// TwinCAT 3 PLC project JobManagement
// Title: JobManagementFramework
// Company: Bekchoff Automation K.K.
// Author: Takashi Ichihashi
// ProjectVersion: 2.0.0.0
// ProgramVersion: 3.1.4026.21
// CompilerDefines: VISU_USEWSTRING, VISU_NO_EXCEPTION_HANDLING
// libraries:
//   CmpBitmapPool, * (System)
//   Tc2_MC2, * (Beckhoff Automation GmbH)
//   Tc2_Standard, * (Beckhoff Automation GmbH)
//   Tc2_System, * (Beckhoff Automation GmbH)
//   Tc2_Utilities, * (Beckhoff Automation GmbH)
//   Tc3_Module, * (Beckhoff Automation GmbH)
// project tree:
//   DUTs/ ContainerType.TcDUT, ErrorTracking.TcDUT, E_ErrorId.TcDUT, E_FutureExecutionState.TcDUT, ST_JobEventMessage.TcDUT, ST_ModuleCylinder2POS.TcDUT, ST_MotionData.TcDUT
//   / GlobalTextList.TcGTLO, PlcTask.TcTTO, Visualization Manager.TcVMO (not stored), VISU_TASK.TcTTO
//   GVLs/ GVL.TcGVL, ParamFuturesLib.TcGVL
//   POUs/ Command.TcDUT, demo1.TcPOU, demo2.TcPOU, demo3.TcPOU, MotionCommand.TcDUT
//   POUs/model/activities/ FB_EventMessageQueue.TcPOU, FutureCounterBlinkCreator.TcPOU, FutureMCGearIn.TcPOU, FutureMCGearInCreator.TcPOU, FutureMCGearOut.TcPOU, FutureMCGearOutCreator.TcPOU, FutureMCHalt.TcPOU, FutureMCHaltCreator.TcPOU, FutureMCInching.TcPOU, FutureMCInchingCreator.TcPOU, FutureMCMoveAbsolute.TcPOU, FutureMCMoveAbsoluteCreator.TcPOU, FutureMCMoveRelative.TcPOU, FutureMCMoveRelativeCreator.TcPOU, FutureMCMoveVelocity.TcPOU, FutureMCMoveVelocityCreator.TcPOU, FutureMCPower.TcPOU, FutureMCPowerCreator.TcPOU, FutureMCReset.TcPOU, FutureMCResetCreator.TcPOU, FutureMCSetPosition.TcPOU, FutureMCSetPositionCreator.TcPOU, FutureMCStop.TcPOU, FutureMCStopCreator.TcPOU, FutureSleep.TcPOU, FutureSleepCreator.TcPOU, FutureTimerBlink.TcPOU, FutureCounterBlink.TcPOU, FutureTimerBlinkCreator.TcPOU
//   POUs/model/library/ FB_AbstructFuture.TcPOU, FB_BatchJobContainer.TcPOU, FB_BatchJobContainerCreator.TcPOU, FB_AbstructContainer.TcPOU, FB_ParallelJobContainerCreator.TcPOU, FB_ParallelQueueJobContainerCreator.TcPOU, FB_QueueJobContainer.TcPOU, FB_Executor.TcPOU, FB_ParallelJobContainer.TcPOU, FB_ParallelQueueJobContainer.TcPOU, FB_QueueJobContainerCreator.TcPOU, FB_TaskRunner.TcPOU, I_Container.TcIO, I_Future.TcIO, I_SerialContainer.TcIO, I_TaskCreator.TcIO, I_Job.TcIO
//   POUs/model/library/Observer/ FB_JobInfoPublisher.TcPOU (not stored), FB_JobEventLogStr.TcPOU, FB_JobEventCyclicOutput.TcPOU, I_JobInfo.TcIO, I_Observer.TcIO, I_Observable.TcIO
//   POUs/test/ FB_TaskRunner_Test.TcPOU, UnitTest.TcPOU
//   VISUs/ ImagePool.TcIPO (not stored), Visualization.TcVIS
// real-time tasks:
//   TASK PlcTask: cycle T#10ms, priority 10, ADS port 350
//   TASK VISU_TASK: cycle T#100000us, priority 12, ADS port 351
// motion (NC):
//   TASK NC-Task 1 SAF: cycle T#1ms, priority 4, ADS port 501
//   TASK NC-Task 1 SVB: cycle T#10ms, priority 8, ADS port 511
//   AXIS Axis 1 (id 1)
//     OtherSettings: AllowMotionCmdToSlave=true
//     encoder EncType=19
//       EncPara: MaxCount=#xffffffff
//     drive DrvType=16
//       DrvPara: MaxCount=#xffffffff
//         Analog: TorqueSetpointScale=10, ScaleFactorActTorque=0.1
//         TimeComp: TaskDelayCycles=1
//     controller CtrType=1
//       CtrPara: PriorControlFactor=1
//         Observer: BandWidth=20
// I/O:
//   DEVICE Device 1 (EtherCAT) (disabled), AmsNetId 199.4.42.250.2.1
//     Term 1 (EK1100) [EK1100 EtherCAT Coupler (2A E-Bus)]
//       Term 2 (EL2008-0015) [EL2008-0015 8Ch. Dig. Output 24V DC, 0.35A, not short-circuit proof]
//       Term 6 (EL2502) [EL2502 2Ch. PWM output, 24V]
//       Term 5 (EL2596) [EL2596 1-channel LED strobe control terminal 24V/3A]
//       Drive 3 (EL7201-9015) [EL7201-9015 1Ch. DS402 Servo motor output stage with OCT (50V, 2.8A RMS) and STO input]
//       Term 4 (EL9011) [EL9011 End Terminal]
//     Term 7 (EC1100) [EC1100 | EtherCAT coupler, RJ45, angled, push-in]
// variable links:
//   JobManagement/JobManagement Instance <-> NC-Task 1 SAF/Axes/Axis 1
//     PlcTask Inputs/GVL.axis1.NcToPlc <-> Outputs/ToPlc
//     PlcTask Outputs/GVL.axis1.PlcToNc <-> Inputs/FromPlc

CONFIGURATION JobManagement
    RESOURCE PLC ON TwinCAT3
        TASK PlcTask(INTERVAL := T#10ms, PRIORITY := 10);
        TASK VISU_TASK(INTERVAL := T#100000us, PRIORITY := 12);
        PROGRAM demo3 WITH PlcTask : demo3;
        PROGRAM VisuElems_Visu_Prg WITH VISU_TASK : VisuElems.Visu_Prg;
    END_RESOURCE
END_CONFIGURATION

// ---- DUTs/ContainerType.TcDUT
{attribute 'qualified_only'}
{attribute 'strict'}
TYPE ContainerType :
(
	BATCH := 0,
	PARALLEL,
	QUEUE,
	PARALLEL_QUEUE
);
END_TYPE

// ---- DUTs/ErrorTracking.TcDUT
TYPE ErrorTracking :
STRUCT
	job_id : STRING;
	error_id : UDINT;
END_STRUCT
END_TYPE

// ---- DUTs/E_ErrorId.TcDUT
{attribute 'qualified_only'}
{attribute 'strict'}
TYPE E_ErrorId :
(
	PASSIVE_ABORT := 16#FFFFFFFF,
	NOT_CONTAINER := 16#FFFFFFFE
) UDINT;
END_TYPE

// ---- DUTs/E_FutureExecutionState.TcDUT
{attribute 'qualified_only'}
{attribute 'strict'}
{attribute 'to_string'}
TYPE E_FutureExecutionState :
(
	idle := 0,
	init,
	wait_for_process,
	process,
	abort,
	pause,
	quit,
	finish
);
END_TYPE

// ---- DUTs/ST_JobEventMessage.TcDUT
{attribute 'pack_mode' := '1'}
TYPE ST_JobEventMessage :
STRUCT
	subject : T_MaxString;
	job_namespace : T_MaxString;
	job_id : T_MaxString;
	old_state : STRING(16);
	new_state : STRING(16);
	num_of_job : UDINT;
	record_time : ULINT; 
END_STRUCT
END_TYPE

// ---- DUTs/ST_ModuleCylinder2POS.TcDUT
TYPE ST_ModuleCylinder2POS :
STRUCT
	in_pos1	AT%I* : BOOL;
	in_pos2	AT%I* : BOOL;
	out_push AT%Q*	: BOOL;
	out_pull AT%Q*	: BOOL;
	timeout_push	: TIME;	
	timeout_pull	: TIME;	
	current_position : E_2Position := E_2Position.pos1; // pos1 : pull side, pos2: push side
END_STRUCT
END_TYPE

// ---- DUTs/ST_MotionData.TcDUT
TYPE ST_MotionData EXTENDS Tc2_MC2.NCTOPLC_AXIS_REF : 
STRUCT
	record_time : ULINT; 
END_STRUCT
END_TYPE

// ---- POUs/Command.TcDUT
{attribute 'qualified_only'}
{attribute 'strict'}
{attribute 'to_string'}
TYPE Command :
(
	spleep := 0,
	power,
	move_absolute,
	move_relative,
	move_velocity
)UDINT;
END_TYPE

// ---- POUs/MotionCommand.TcDUT
TYPE MotionCommand :
STRUCT
	activate	: BOOL;
	command_id	: Command;
	target		: LREAL;
	velocity	: LREAL;
END_STRUCT
END_TYPE

// ---- GVLs/GVL.TcGVL
{attribute 'qualified_only'}
VAR_GLOBAL
	batch_job_container_creator : FB_BatchJobContainerCreator;
	parallel_job_container_creator : FB_ParallelJobContainerCreator;
	queue_job_container_creator : FB_QueueJobContainerCreator;
	parallel_queue_job_container_creator : FB_ParallelQueueJobContainerCreator;
	axis1	: AXIS_REF;
	axis2	: AXIS_REF;
	motion_command : MotionCommand;
END_VAR

// ---- GVLs/ParamFuturesLib.TcGVL
{attribute 'qualified_only'}
VAR_GLOBAL CONSTANT
	MAX_TASK_NUM : UINT := 40; // Number of max jobs in job container object.
	MAX_STRING_LENGTH : UDINT := 255; // Max string length of task name.
END_VAR

// ---- POUs/model/library/I_Container.TcIO
INTERFACE I_Container EXTENDS __SYSTEM.IQueryInterface

(* This is the generator that iteratively generates references to FB_executor instances*)
METHOD _index_generator_ : UINT;
VAR_INPUT
END_VAR
END_METHOD

METHOD append_job : I_Job
VAR_INPUT
	executor	: I_Job;
END_VAR
END_METHOD

PROPERTY auto_start : BOOL
GET
END_GET
SET
END_SET
END_PROPERTY

PROPERTY continuous_mode : bool
SET
END_SET
END_PROPERTY

METHOD create_container : I_Job
VAR_INPUT
	container_type : ContainerType;
	name: STRING;
END_VAR
END_METHOD

METHOD create_job : I_Job
VAR_INPUT
	creator : I_TaskCreator;
	future_name: STRING;
END_VAR
END_METHOD

PROPERTY each_executor : I_Job
GET
END_GET
END_PROPERTY

PROPERTY num_of_jobs : UDINT
GET
END_GET
END_PROPERTY

METHOD reset : BOOL // Return TRUE if finish.
VAR_INPUT
	deep : BOOL := FALSE;
END_VAR
END_METHOD

METHOD resume : BOOL
VAR_INPUT
END_VAR
END_METHOD

METHOD spawn_job : I_Job
VAR_INPUT
	future : I_Future;
	job_persistence : BOOL := FALSE;
END_VAR
END_METHOD

END_INTERFACE

// ---- POUs/model/library/I_Future.TcIO
{attribute 'enable_dynamic_creation'}
INTERFACE I_Future EXTENDS __System.IQueryInterface

METHOD abort : BOOL // Return TRUE if finish.
VAR_INPUT
END_VAR
END_METHOD

METHOD error_reset : BOOL
VAR_INPUT
END_VAR
END_METHOD

METHOD execute : BOOL // Return TRUE if finish.
VAR_INPUT
END_VAR
END_METHOD

PROPERTY executor : I_Job
GET
END_GET
SET
END_SET
END_PROPERTY

PROPERTY future_name : STRING // Name of future.
GET
END_GET
SET
END_SET
END_PROPERTY

METHOD init : BOOL // Return TRUE if finish.
VAR_INPUT
END_VAR
END_METHOD

PROPERTY nErrorID : HRESULT // Set result code when finished any method. 0 should be set when normal case.
GET
END_GET
END_PROPERTY

PROPERTY persistent_future : BOOL
GET
END_GET
SET
END_SET
END_PROPERTY

METHOD quit : BOOL // Return TRUE if finish.
VAR_INPUT
END_VAR
END_METHOD

PROPERTY state : E_FutureExecutionState // Execution state of this future.
GET
END_GET
SET
END_SET
END_PROPERTY

END_INTERFACE

// ---- POUs/model/library/I_SerialContainer.TcIO
INTERFACE I_SerialContainer EXTENDS __SYSTEM.IQueryInterface

PROPERTY current_job : I_Job
GET
END_GET
END_PROPERTY

END_INTERFACE

// ---- POUs/model/library/I_TaskCreator.TcIO
INTERFACE I_TaskCreator

METHOD create_future : I_Future
VAR_INPUT
	future_name :STRING; // Specify future name
END_VAR
END_METHOD

METHOD destroy_future : I_Future
VAR_INPUT
	future : I_Future; // Specify future instance whtat you want to delete.
END_VAR
END_METHOD

END_INTERFACE

// ---- POUs/model/library/I_Job.TcIO
INTERFACE I_Job EXTENDS __SYSTEM.IQueryInterface

(*abort method

*)
METHOD abort : BOOL // Return TRUE if finish.
VAR_INPUT
END_VAR
END_METHOD

PROPERTY busy : BOOL
GET
END_GET
END_PROPERTY

PROPERTY children : I_Container // Accesser for interface pointer to child container instance.
GET
END_GET
END_PROPERTY

PROPERTY continuous_mode : bool // Make true if keep executing state after all jobs be finished.
SET
END_SET
END_PROPERTY

METHOD create_container : I_Container // Make container object onto child.
VAR_INPUT
	container_type : ContainerType; // specify container type
	name: STRING;	// specify future name
END_VAR
END_METHOD

METHOD create_future : I_Future // Create future dynamically.
VAR_INPUT
	creator : I_TaskCreator; // Specify creator object by which Interface Task Creator implemented.
	future_name: STRING; // Spcfigy future name.
END_VAR
END_METHOD

{attribute 'OPC.UA.DA.Property' := '1'}
{attribute 'monitoring' := 'call'}
{attribute 'OPC.UA.DA.Description' := 'Current state of this executor object.'}
PROPERTY current_state : E_FutureExecutionState // Get current job state
GET
END_GET
END_PROPERTY

PROPERTY current_timestamp : POINTER TO T_FILETIME64
GET
END_GET
SET
END_SET
END_PROPERTY

PROPERTY done : BOOL // Present true if process be finished.
GET
END_GET
END_PROPERTY

METHOD error_reset : BOOL
VAR_INPUT
END_VAR
END_METHOD

METHOD execute : BOOL // Execute future process and return TRUE if all task are finished.
END_METHOD

PROPERTY future : I_Future // Set future instance direct.
GET
END_GET
SET
END_SET
END_PROPERTY

PROPERTY future_creator : I_TaskCreator // Set creator instance.
SET
END_SET
END_PROPERTY

METHOD get_job_info : BOOL
VAR_INPUT
	title		: T_MaxString;
	observable 	: I_Observable;
	recursive	: BOOL := FALSE;
END_VAR
END_METHOD

PROPERTY id : T_MaxString // Get job id.
GET
END_GET
END_PROPERTY

METHOD init : BOOL // Return TRUE if finish.
VAR_INPUT
END_VAR
END_METHOD

PROPERTY job_event_observable : I_Observable
GET
END_GET
SET
END_SET
END_PROPERTY

PROPERTY last_state : E_FutureExecutionState
GET
END_GET
END_PROPERTY

PROPERTY namespace : T_MaxString
GET
END_GET
END_PROPERTY

PROPERTY nErrorID : HRESULT // Present error code when each process,init(), execute(), quit() are finished. '0' represent normal condition without any errors.
GET
END_GET
END_PROPERTY

PROPERTY next_job : I_Job
GET
END_GET
SET
END_SET
END_PROPERTY

PROPERTY parent_executor : I_Job
GET
END_GET
SET
END_SET
END_PROPERTY

PROPERTY persistent_job : BOOL
GET
END_GET
SET
END_SET
END_PROPERTY

PROPERTY previous_job : I_Job
GET
END_GET
SET
END_SET
END_PROPERTY

METHOD quit : BOOL // Return TRUE if finish.
VAR_INPUT
END_VAR
END_METHOD

PROPERTY ready : BOOL
GET
END_GET
END_PROPERTY

METHOD reset : BOOL // Return TRUE if finish.
VAR_INPUT
	deep : BOOL := FALSE;
END_VAR
END_METHOD

METHOD resume : BOOL
END_METHOD

PROPERTY serial : ULINT
GET
END_GET
SET
END_SET
END_PROPERTY

METHOD start : BOOL
END_METHOD

PROPERTY transition : BOOL
GET
END_GET
END_PROPERTY

PROPERTY upstream_aborting : BOOL
GET
END_GET
SET
END_SET
END_PROPERTY

END_INTERFACE

// ---- POUs/model/library/Observer/I_JobInfo.TcIO
INTERFACE I_JobInfo EXTENDS __SYSTEM.IQueryInterface

PROPERTY job : I_Job
GET
END_GET
SET
END_SET
END_PROPERTY

PROPERTY last_state : E_FutureExecutionState
GET
END_GET
SET
END_SET
END_PROPERTY

PROPERTY new_state : E_FutureExecutionState
GET
END_GET
SET
END_SET
END_PROPERTY

PROPERTY record_time : T_FILETIME64
GET
END_GET
SET
END_SET
END_PROPERTY

PROPERTY title : T_MaxString
GET
END_GET
SET
END_SET
END_PROPERTY

END_INTERFACE

// ---- POUs/model/library/Observer/I_Observer.TcIO
INTERFACE I_Observer

METHOD notify : BOOL
VAR_INPUT
	publisher : I_Observable;
END_VAR
END_METHOD

END_INTERFACE

// ---- POUs/model/library/Observer/I_Observable.TcIO
INTERFACE I_Observable  EXTENDS __SYSTEM.IQueryInterface

METHOD add_observer : BOOL
VAR_INPUT
	observer : I_Observer;
END_VAR
END_METHOD

PROPERTY error_id : HRESULT
GET
END_GET
SET
END_SET
END_PROPERTY

METHOD notify_observers : BOOL
END_METHOD

METHOD remove_observer : BOOL
VAR_INPUT
	observer : I_Observer;
END_VAR
END_METHOD

END_INTERFACE

// ---- POUs/demo3.TcPOU
PROGRAM demo3
VAR
	runner : FB_TaskRunner(ContainerType.PARALLEL_QUEUE);

	init: BOOL;
	_state :UINT;
	mc_power : FutureMCPower;
	_handl_power_on	: I_Job;
	_handl_demo_job : I_Job;
	
	_today : TIMESTRUCT;

	bPower : BOOL;
	bStart : BOOL;

	motion_data : ST_MotionData;	
	demo_job_container : FB_BatchJobContainer;
	i : UDINT;
END_VAR

IF NOT init THEN
	JobCreateDemo(demo_job_container, GVL.axis1); // demo_job にメソッドを通してシーケンスジョブを組み立てる
	mc_power.future_name := 'POWER_CTRL';
	init := TRUE;	// RUN 後 1 サイクルだけ実行
END_IF

_today := FILETIME64_TO_SYSTEMTIME(runner.current_time);
runner(root_job_name := 'ROOT',root_job_serial := (_today.wYear MOD 100) * 10000 + _today.wMonth * 100 + _today.wDay);

// Axis
GVL.axis1.ReadStatus();
MEMCPY(ADR(motion_data), ADR(GVL.axis1.NcToPlc), SIZEOF(GVL.axis1.NcToPlc));
motion_data.record_time := runner.current_time;

CASE _state OF
	0:
		IF bPower THEN
			mc_power.set_parameters(axis := GVL.axis1, status := TRUE); // Servo on
			_handl_power_on := runner.append_future(mc_power);
			_state := 1;
		END_IF
	1:
		IF _handl_power_on.ready THEN
			_handl_power_on.start();
		END_IF
		IF _handl_power_on.done THEN
			_state := 2;
		END_IF
	2:
		IF bStart THEN
			_handl_demo_job := runner.append_future(demo_job_container);
			_state := 3;
		END_IF
	3:
		IF _handl_demo_job.ready THEN
			_handl_demo_job.start();
		END_IF
		IF _handl_demo_job.current_state = E_FutureExecutionState.finish THEN
			_state := 2;
			//bStart := FALSE;
		END_IF
		IF NOT bPower THEN
			_state := 4;
		END_IF
	4:
		IF runner.halt(_handl_demo_job) THEN
			_state := 5;
		END_IF
	5:
		mc_power.set_parameters(axis := GVL.axis1, status := FALSE); // Servo off
		_handl_power_on := runner.append_future(mc_power);
		_state := 6;
	6:
		IF _handl_power_on.ready THEN
			_handl_power_on.start();
		END_IF
		IF _handl_power_on.done THEN
			_state := 0;
		END_IF
END_CASE

//IF _state > 0 AND NOT bPower THEN
//END_IF

METHOD JobCreateDemo : BOOL
VAR_INPUT
	job_container : I_Container;
	stAxis1	: REFERENCE TO AXIS_REF;
END_VAR
VAR
	_base_future : I_Future;
	_job_temp : I_Job;
	_job_temp_parent : I_Job;
	sleep : POINTER TO FutureSleep;
	sleep_creator : FutureSleepCreator;

	//mc_move_rel_future : POINTER TO FutureMCMoveRelative;
	mc_move_rel_future_creator : FutureMCMoveRelativeCreator;

	//mc_move_abs_future : POINTER TO FutureMCMoveAbsolute;
	mc_move_abs_future_creator : FutureMCMoveAbsoluteCreator;

	//mc_move_velocity_future: POINTER TO FutureMCMoveVelocity;
	mc_move_velocity_future_creator: FutureMCMoveVelocityCreator;
	
	mc_stop_future_creator : FutureMcStopCreator;
	
	i : UDINT;

END_VAR
//base_job.create_container(ContainerTYpe.BATCH, 'DEMO_JOB');
IF __QUERYINTERFACE(job_container,_base_future) THEN
	_base_future.future_name := 'JOB ROOT';
END_IF

// Sequence
_job_temp_parent := job_container.create_container(ContainerTYpe.BATCH, 'STEP MOVING');
FOR i := 1 TO 4 DO

	mc_move_rel_future_creator.set_parameters(stAxis1,20,200,0,0,0,0);
	_job_temp := _job_temp_parent.children.create_job(mc_move_rel_future_creator,'Move +20 deg, 200 deg/s');

	sleep_creator.sleep_time := T#100MS;
	_job_temp := _job_temp_parent.children.create_job(sleep_creator,'Wait 100ms');
	
END_FOR

// position set to 0

mc_move_abs_future_creator.set_parameters(stAxis1,0,200,0,0,0,0);
_job_temp := job_container.create_job(mc_move_abs_future_creator,'Back to home');

FOR i := 1 TO 10 DO

	mc_move_rel_future_creator.set_parameters(stAxis1,-20,200,0,0,0,0);
	_job_temp := job_container.create_job(mc_move_rel_future_creator,'Move -20 deg, 200 deg/s');

	sleep_creator.sleep_time := T#100MS;
	_job_temp := job_container.create_job(sleep_creator,'Wait 100ms');
	
END_FOR

// position to 0

mc_move_abs_future_creator.set_parameters(stAxis1,0,200,0,0,0,0);
_job_temp := job_container.create_job(mc_move_abs_future_creator,'Back to home');

sleep_creator.sleep_time := T#100MS;
_job_temp := job_container.create_job(sleep_creator,'Wait 100ms');

// 1000deg/s -> 500deg/s

mc_move_velocity_future_creator.set_parameters(stAxis1,MC_Direction.MC_Positive_Direction,10,0,0,0,0);
_job_temp := job_container.create_job(mc_move_velocity_future_creator,'Move velocity');

sleep_creator.sleep_time := T#5S;
_job_temp := job_container.create_job(sleep_creator,'10 deg/s 5 seconds');

mc_move_velocity_future_creator.set_parameters(stAxis1,MC_Direction.MC_Positive_Direction,100,0,0,0,0);
_job_temp := job_container.create_job(mc_move_velocity_future_creator,'Move velocity');

sleep_creator.sleep_time := T#5S;
_job_temp := job_container.create_job(sleep_creator,'100 deg/s 5 seconds');

mc_move_velocity_future_creator.set_parameters(stAxis1,MC_Direction.MC_Positive_Direction,250,0,0,0,0);
_job_temp := job_container.create_job(mc_move_velocity_future_creator,'Move velocity');

sleep_creator.sleep_time := T#5S;
_job_temp := job_container.create_job(sleep_creator,'250 deg/s 5 seconds');

mc_stop_future_creator.set_parameters(stAxis1,0,0);
_job_temp := job_container.create_job(mc_stop_future_creator,'STOP');

// position to 0

mc_move_abs_future_creator.set_parameters(stAxis1,0,250,0,0,0,0);
_job_temp := job_container.create_job(mc_move_abs_future_creator,'Back to home');
END_METHOD

END_PROGRAM

// ---- POUs/model/library/FB_TaskRunner.TcPOU
FUNCTION_BLOCK FB_TaskRunner
VAR_INPUT
	error_reset : BOOL; // Error reset
	root_job_serial : ULINT := 1;
	root_job_name : STRING := 'ROOT';
	upstream_aborting : BOOL := FALSE; // 
	continuous_mode : BOOL := TRUE;
END_VAR
VAR_OUTPUT
	job_empty : BOOL;
	job_namespace : T_MaxString;
	num_of_jobs : UDINT;
END_VAR
VAR
	_executor: FB_Executor; // main Executor
	_observable : FB_JobInfoPublisher;
	last_job_number : UDINT;
	job_event_log_str : FB_JobEventLogStr;	// ジョブイベントをメッセージとしてログ出力するサブスクライバ
	job_event_cyclic_output : FB_JobEventCyclicOutput;	// ADS通信向けにジョブイベントをサイクル単位で出力するためのサブスクライバ
	
	
	fbGetTimeZoneInformation	: FB_GetTimeZoneInformation := (bExecute := TRUE);
	localTime : FB_LocalSystemTime := (bEnable := TRUE);
	tzinfo : FB_GetTimeZoneInformation := (bExecute := TRUE);
	getSystemtime : FB_TzSpecificLocalTimeToSystemTime;
	_current_time : T_FILETIME64;
END_VAR

// 現在時刻の取得
localTime();
tzinfo();
getSystemtime(in := localTime.systemTime, tzInfo := tzinfo.tzInfo);
_current_time := SYSTEMTIME_TO_FILETIME64(getSystemtime.out);
_executor.current_timestamp := ADR(_current_time);

// Job event log for ADS output 
job_event_cyclic_output(); 

_executor.serial := root_job_serial;
_executor.execute();
num_of_jobs := _executor.children.num_of_jobs;

job_empty := last_job_number > 0 AND _executor.children.num_of_jobs = 0;
last_job_number := _executor.children.num_of_jobs;


IF _executor.ready THEN
	_executor.start();
END_IF

METHOD abort : BOOL
VAR_INPUT
	job : I_Job := 0;
END_VAR
VAR
	_child_executor : I_Job;
	all_aborted : BOOL;
END_VAR
IF _executor.children = 0 THEN
	abort := TRUE;
	RETURN;
END_IF

//IF job = 0 OR num_of_jobs = 0 THEN
	all_aborted := TRUE;
//END_IF
REPEAT
	_child_executor := _executor.children.each_executor;
	IF _child_executor <> 0 THEN
		IF job <> 0 THEN
			IF job = _child_executor THEN
				all_aborted := _child_executor.abort();
			END_IF
		ELSE
			IF NOT _child_executor.abort() THEN
				all_aborted := FALSE;
			END_IF
		END_IF

	END_IF
UNTIL
	_child_executor = 0
END_REPEAT

abort := all_aborted;
END_METHOD

METHOD append_future : I_Job
VAR_INPUT
	future : I_Future;
END_VAR
IF _executor.children = 0 THEN
	RETURN;
END_IF

append_future := _executor.children.spawn_job(future, TRUE);
job_namespace := append_future.namespace;
END_METHOD

METHOD append_job : I_Job
VAR_INPUT
	job : I_Job;
END_VAR
IF _executor.children = 0 THEN
	append_job := 0;
	RETURN;
END_IF

append_job := _executor.children.append_job(job);
job_namespace := append_job.namespace;
END_METHOD

METHOD create_job : I_Job
VAR_INPUT
	creator : I_TaskCreator;
	name : STRING;
END_VAR
IF _executor.children = 0 THEN
	RETURN;
END_IF

create_job := _executor.children.create_job(creator, name);
job_namespace := create_job.namespace;
END_METHOD

PROPERTY current_time : T_FILETIME64
GET
current_time := _current_time;
END_GET
END_PROPERTY

METHOD error_reset : BOOL
VAR_INPUT
END_VAR
error_reset := _executor.error_reset();
END_METHOD

//FB_Init is always available implicitly and it is used primarily for initialization.
//The return value is not evaluated. For a specific influence, you can also declare the
//methods explicitly and provide additional code there with the standard initialization
//code. You can evaluate the return value.
METHOD FB_Init: BOOL
VAR_INPUT
    bInitRetains: BOOL; // TRUE: the retain variables are initialized (reset warm / reset cold)
    bInCopyCode: BOOL;  // TRUE: the instance will be copied to the copy code afterward (online change)
	container_type : ContainerType := ContainerType.QUEUE;
END_VAR
_executor.job_event_observable := _observable;
_observable.add_observer(job_event_log_str);
_observable.add_observer(job_event_cyclic_output);
_executor.upstream_aborting := upstream_aborting;
_executor.create_container(container_type, root_job_name);
_executor.continuous_mode := TRUE;
END_METHOD

METHOD halt : BOOL
VAR_INPUT
	job : I_Job;
END_VAR
IF job <> 0 AND_THEN NOT job.done THEN
	IF THIS^.abort(job) THEN
		IF THIS^.quit(job) THEN
			IF THIS^.job_clear(job) THEN
				halt := TRUE;
			END_IF
		END_IF
	END_IF
END_IF
END_METHOD

METHOD job_clear : BOOL
VAR_INPUT
	job : I_Job := 0;
END_VAR
VAR
	_child_executor : I_Job;
	all_clear : BOOL;
	
END_VAR
IF _executor.children = 0 THEN
	job_clear := TRUE;
	RETURN;
END_IF

job_clear := _executor.children.reset(FALSE);
END_METHOD

PROPERTY job_event_observable : I_Observable
GET
job_event_observable := _executor.job_event_observable;
END_GET
SET
_executor.job_event_observable := job_event_observable;
END_SET
END_PROPERTY

METHOD quit : BOOL
VAR_INPUT
	job : I_Job := 0;
END_VAR
VAR
	_child_executor : I_Job;
	all_quit: BOOL;
END_VAR
IF _executor.children = 0 THEN
	quit := TRUE;
	RETURN;
END_IF

//IF job = 0 OR _executor.children.num_of_jobs > 0 THEN
	all_quit := TRUE;
//END_IF

REPEAT
	_child_executor := _executor.children.each_executor;
	IF _child_executor <> 0 THEN
		IF job <> 0 THEN
			IF job = _child_executor THEN
				all_quit := _child_executor.quit();
			END_IF
		ELSE
			IF NOT _child_executor.quit() THEN
				all_quit := FALSE;
			END_IF
		END_IF

	END_IF
UNTIL
	_child_executor = 0
END_REPEAT

quit := all_quit;
END_METHOD

METHOD restart : BOOL
VAR_INPUT
END_VAR
IF _executor.error_reset() THEN
	restart := _executor.resume();
END_IF
END_METHOD

PROPERTY root_executor : I_Job
GET
root_executor := _executor;
END_GET
END_PROPERTY

END_FUNCTION_BLOCK

// ---- POUs/model/library/FB_Executor.TcPOU
{attribute 'enable_dynamic_creation'}
FUNCTION_BLOCK FB_Executor IMPLEMENTS I_Job
VAR_INPUT
END_VAR
VAR_OUTPUT
END_VAR
VAR
	{attribute 'TcEncoding':='UTF-8'}
	_namespace : T_MaxString;
	_id : T_MaxString;
	_done : BOOL;
	_start : BOOL;
	_resume : BOOL;
	_passive_abort : BOOL;
	_quit : BOOL;
	_upstream_aborting : BOOL := FALSE;
	 {attribute 'TcAnalytics'}
	 _state :E_FutureExecutionState := E_FutureExecutionState.idle;
	_last_state  :E_FutureExecutionState;
	_error_id : HRESULT;
	_aborting :BOOL;
	_quitting :BOOL;
	_interface_container : I_Container := 0;
	_job_event_observable : I_Observable;
	_future_creator : I_TaskCreator;
	_future : I_Future;
	_parent_job : I_Job := 0;
	_persistent_job : BOOL := TRUE;
	_current_timestamp : POINTER TO T_FILETIME64 := 0;
	_previous_job : I_Job;
	_next_job : I_Job;
	_transition : BOOL;
END_VAR
VAR PERSISTENT
	_serial	: ULINT;
END_VAR

(*abort method

*)
METHOD abort : BOOL // Return TRUE if finish.
VAR_INPUT
END_VAR
IF _state = E_FutureExecutionState.init OR
   _state = E_FutureExecutionState.process OR
   _state = E_FutureExecutionState.quit THEN
   	_start := FALSE;
	_passive_abort := TRUE;
	abort := FALSE;
ELSE
	IF _state = E_FutureExecutionState.abort THEN
		abort := NOT _aborting;
	ELSE
		abort := TRUE;
	END_IF
END_IF
THIS^.execute();
END_METHOD

PROPERTY busy : BOOL
GET
busy := (	_state = E_FutureExecutionState.init OR	
			_state = E_FutureExecutionState.process OR 
			_state = E_FutureExecutionState.quit
		);
END_GET
END_PROPERTY

PROPERTY children : I_Container // Accesser for interface pointer to child container instance.
GET
children := _interface_container;
END_GET
END_PROPERTY

PROPERTY continuous_mode : bool // Make true if keep executing state after all jobs be finished.
SET
IF _interface_container <> 0 THEN
	_interface_container.continuous_mode := continuous_mode;
END_IF
END_SET
END_PROPERTY

METHOD create_container : I_Container // Make container object onto child.
VAR_INPUT
	container_type : ContainerType; // specify container type
	name: STRING;	// specify future name
END_VAR
VAR
	delete_existing_container : BOOL;
	created_future : I_Future;
END_VAR
IF _interface_container <> 0 THEN
 	IF _interface_container.reset(FALSE) THEN
		delete_existing_container := TRUE;
	ELSE
		delete_existing_container := FALSE;
	END_IF
ELSE
	delete_existing_container := TRUE;
END_IF

IF delete_existing_container THEN
	CASE container_type OF
		ContainerType.BATCH:
			created_future := create_future(GVL.batch_job_container_creator, name);
			created_future.executor.persistent_job := FALSE;
		ContainerType.PARALLEL:
			created_future := create_future(GVL.parallel_job_container_creator, name);
			created_future.executor.persistent_job := FALSE;
		ContainerType.QUEUE:
			created_future := create_future(GVL.queue_job_container_creator, name);
			created_future.executor.persistent_job := TRUE;
		ContainerType.PARALLEL_QUEUE:
			created_future := create_future(GVL.parallel_queue_job_container_creator, name);
			created_future.executor.persistent_job := TRUE;
	END_CASE
	THIS^.init();
	create_container := THIS^.children;
END_IF
END_METHOD

METHOD create_future : I_Future // Create future dynamically.
VAR_INPUT
	creator : I_TaskCreator; // Specify creator object by which Interface Task Creator implemented.
	future_name: STRING; // Spcfigy future name.
END_VAR
_future_creator := creator;
IF _future_creator <> 0 THEN
	THIS^.future := creator.create_future(future_name);
	_future.persistent_future := FALSE;
END_IF
create_future := _future;
END_METHOD

{attribute 'OPC.UA.DA.Property' := '1'}
{attribute 'monitoring' := 'call'}
{attribute 'OPC.UA.DA.Description' := 'Current state of this executor object.'}
PROPERTY current_state : E_FutureExecutionState // Get current job state
GET
current_state := _state;
END_GET
END_PROPERTY

PROPERTY current_timestamp : POINTER TO T_FILETIME64
GET
current_timestamp := _current_timestamp;
END_GET
SET
_current_timestamp := current_timestamp;
END_SET
END_PROPERTY

PROPERTY done : BOOL // Present true if process be finished.
GET
done := _done;
END_GET
END_PROPERTY

METHOD error_reset : BOOL
VAR_INPUT
END_VAR
IF _future <> 0 THEN
	IF _future.error_reset() THEN
		error_reset := TRUE;
		get_job_info('ERROR_RESET', _job_event_observable, FALSE);
	ELSE
		error_reset := FALSE;
	END_IF
	_error_id := _future.nErrorID;
ELSE
	_error_id := 0;
	error_reset := TRUE;
END_IF
END_METHOD

METHOD execute : BOOL // Execute future process and return TRUE if all task are finished.
VAR_INST
	_state_mem :E_FutureExecutionState;
	delay : TIME := T#3S;
	sleep : TON;
	await : BOOL;
	_logging : BOOL;
END_VAR
VAR
	_executor : REFERENCE TO FB_Executor;
	start_all_children : BOOL;
	exe: INT;
END_VAR
IF _future = 0 THEN
	execute := TRUE;
	RETURN;
ELSE
	execute := FALSE;
END_IF

IF _passive_abort THEN
	_state := E_FutureExecutionState.abort;
	//IF _error_id = 0 THEN
	//	_error_id := E_ErrorId.PASSIVE_ABORT;
	//END_IF
	_passive_abort := FALSE;
END_IF

IF _quit THEN
	_state := E_FutureExecutionState.quit;
END_IF
_quit := FALSE;

CASE _state OF
	E_FutureExecutionState.idle:
		IF _future.state = E_FutureExecutionState.idle OR 
			_future.state = E_FutureExecutionState.finish THEN
			IF init() THEN
				_state := E_FutureExecutionState.init;
			END_IF
		END_IF
	E_FutureExecutionState.init:
		IF _future.init() THEN
			IF _future.nErrorID = 0 THEN
				_state := E_FutureExecutionState.wait_for_process;
			ELSE
				_last_state := E_FutureExecutionState.init;
				_error_id := _future.nErrorID;
				_state := E_FutureExecutionState.abort;
			END_IF
		END_IF
	E_FutureExecutionState.wait_for_process: 
		IF _start THEN
			IF _previous_job <> 0 AND_THEN _future <> 0 AND_THEN _previous_job.future = _future THEN
				IF _future.init() THEN
					_state := E_FutureExecutionState.process;
					_start := FALSE;					
				END_IF
			ELSE
				_state := E_FutureExecutionState.process;
				_start := FALSE;
			END_IF
		END_IF
	E_FutureExecutionState.process: 
		IF _future.execute() THEN
			IF _future.nErrorID = 0 THEN
				_state := E_FutureExecutionState.quit;
				_done := TRUE;
			ELSE
				_error_id := _future.nErrorID;
				_state := E_FutureExecutionState.abort;
			END_IF
		END_IF
	E_FutureExecutionState.abort:
		IF _aborting THEN
			await := _future.abort();
			_resume := FALSE;
			IF _upstream_aborting AND _parent_job <> 0 THEN
				_parent_job.abort();
			END_IF
			IF await THEN
				_aborting := FALSE;
			END_IF
		ELSIF _resume THEN
			_state := _last_state;
			IF _error_id = E_ErrorId.PASSIVE_ABORT THEN
				_error_id := 0;
			END_IF
			_resume := FALSE;
		END_IF
	E_FutureExecutionState.quit:
		IF _future.quit() THEN
			IF _future.nErrorID = 0 THEN
				_state := E_FutureExecutionState.finish;
			ELSE
				_error_id := _future.nErrorID;
				_state := E_FutureExecutionState.abort;
			END_IF
			_quitting := FALSE;
		END_IF
	E_FutureExecutionState.finish:
		IF NOT _logging THEN
			execute := TRUE;
		END_IF
END_CASE

IF _state <> _state_mem THEN
	_last_state := _state_mem;

	IF _state = E_FutureExecutionState.init OR
		_state = E_FutureExecutionState.process OR
		_state = E_FutureExecutionState.quit THEN
		_error_id := 0;
	END_IF

	IF _state = E_FutureExecutionState.abort THEN
		_aborting := TRUE;
	END_IF
	
	IF _state = E_FutureExecutionState.quit THEN
		sleep(IN := FALSE);
		_quitting := TRUE;
	END_IF

	_logging := TRUE;

END_IF

_transition := _state <> _state_mem;
_state_mem := _state;

// Transition logging
IF _logging THEN
	IF get_job_info('TRANSITION', _job_event_observable,FALSE) THEN
		_logging := FALSE;
	END_IF
END_IF



IF _future <> 0 THEN
	_future.state := _state;
END_IF
END_METHOD

PROPERTY future : I_Future // Set future instance direct.
GET
future := _future;
END_GET
SET
VAR
	_eval_executor : I_Job;
END_VAR
_future := future;
_future.state := _state;
_future.executor := THIS^;
//_future.persistent_future := TRUE;
IF NOT __QUERYINTERFACE(_future, _interface_container) THEN
	_interface_container := 0;
END_IF

_future.persistent_future := TRUE;

// Redefine parent job pointer to the container members which has been set as the new future.
IF _interface_container <> 0 THEN
	REPEAT
		_eval_executor := _interface_container.each_executor;
		IF _eval_executor <> 0 THEN
			// Set persistent future flag when redefine new parent due to make bound of namespace.
			//IF _eval_executor.parent_executor = 0 AND _eval_executor.children <> 0 THEN
			//	_eval_executor.future.persistent_future := TRUE;
			//END_IF
			// Set new parent for each childrens
			_eval_executor.parent_executor := THIS^;
		END_IF
	UNTIL
		_eval_executor = 0
	END_REPEAT
END_IF
END_SET
END_PROPERTY

PROPERTY future_creator : I_TaskCreator // Set creator instance.
SET
_future_creator := future_creator;
END_SET
END_PROPERTY

METHOD get_job_info : BOOL
VAR_INPUT
	title		: T_MaxString; // Observable object title
	observable 	: I_Observable; // Observable object
	recursive	: BOOL := FALSE; // Set observable to child job recursively or not
END_VAR
VAR
	_info : I_JobInfo;
	_child_job : I_Job;
	_cmp : BOOL;
END_VAR
IF observable = 0  OR NOT __QUERYINTERFACE(observable, _info) THEN
	get_job_info := TRUE;
	RETURN;
END_IF

_info.title := title;
_info.job := THIS^;
_info.last_state := _last_state;
_info.new_state := _state;
IF _current_timestamp <> 0 THEN
	_info.record_time := _current_timestamp^;
ELSE
	_info.record_time := F_GetSystemTime();
END_IF

observable.notify_observers();

IF recursive THEN
	_cmp := TRUE;
	IF THIS^.children <> 0 THEN
		REPEAT
			_child_job := THIS^.children.each_executor;
			IF _child_job <> 0 THEN
				IF NOT _child_job.get_job_info(title, observable, recursive) THEN
					_cmp := FALSE;
				END_IF
			END_IF
		UNTIL
			_child_job = 0
		END_REPEAT
	END_IF
	
	get_job_info := _cmp;
ELSE
	get_job_info := TRUE;
END_IF
END_METHOD

PROPERTY id : T_MaxString // Get job id.
GET
id := _id;
END_GET
END_PROPERTY

METHOD init : BOOL // Return TRUE if finish.
VAR_INPUT
END_VAR
VAR
	_eval_executor : I_Job;
END_VAR
_done := FALSE;
_passive_abort := FALSE;
_start := FALSE;
_state := E_FutureExecutionState.idle;
_error_id := 0;

_eval_executor := _parent_job;
_id := CONCAT('/', TO_STRING(_serial));
REPEAT
	IF _eval_executor <> 0 THEN
		_id := CONCAT(TO_STRING(_eval_executor.serial), _id);
		_id := CONCAT('/',_id);
		_eval_executor := _eval_executor.parent_executor;
	END_IF
UNTIL
	_eval_executor = 0
END_REPEAT


IF _parent_job = 0 THEN
	_namespace := _id;
ELSIF _future <> 0 AND_THEN _future.persistent_future AND_THEN NOT _parent_job.future.persistent_future THEN
	_namespace := _id;
ELSE
	_namespace := _parent_job.namespace;
END_IF

INIT := TRUE;
END_METHOD

PROPERTY job_event_observable : I_Observable
GET
job_event_observable := _job_event_observable;
END_GET
SET
VAR
	executor : I_Job;
END_VAR
_job_event_observable := job_event_observable;
IF THIS^.children <> 0 THEN
	REPEAT
		executor := THIS^.children.each_executor;
		IF executor <> 0 THEN
			executor.job_event_observable := job_event_observable;
		END_IF
	UNTIL
		executor = 0
	END_REPEAT
END_IF
END_SET
END_PROPERTY

PROPERTY last_state : E_FutureExecutionState
GET
last_state := _last_state;
END_GET
END_PROPERTY

PROPERTY namespace : T_MaxString
GET
namespace := _namespace;
END_GET
END_PROPERTY

PROPERTY nErrorID : HRESULT // Present error code when each process,init(), execute(), quit() are finished. '0' represent normal condition without any errors.
GET
nErrorID := _error_id;
END_GET
END_PROPERTY

PROPERTY next_job : I_Job
GET
next_job := _next_job;
END_GET
SET
_next_job := next_job;
END_SET
END_PROPERTY

PROPERTY parent_executor : I_Job
GET
parent_executor := _parent_job;
END_GET
SET
VAR
END_VAR
VAR
	_parent_path : T_MaxString;
END_VAR
_parent_job := parent_executor;
THIS^.current_timestamp := _parent_job.current_timestamp;
END_SET
END_PROPERTY

PROPERTY persistent_job : BOOL
GET
persistent_job := _persistent_job;
END_GET
SET
_persistent_job := persistent_job;
END_SET
END_PROPERTY

PROPERTY previous_job : I_Job
GET
previous_job := _previous_job;
END_GET
SET
_previous_job := previous_job;
END_SET
END_PROPERTY

METHOD quit : BOOL // Return TRUE if finish.
VAR_INPUT
END_VAR
IF _state = E_FutureExecutionState.init OR
   _state = E_FutureExecutionState.process OR
   _state = E_FutureExecutionState.quit THEN
	_quit := TRUE;	
END_IF

IF 	_quit AND _state = E_FutureExecutionState.quit THEN
	quit := NOT _quitting;
ELSE
	quit := TRUE;
END_IF
END_METHOD

PROPERTY ready : BOOL
GET
ready := _state = E_FutureExecutionState.wait_for_process;
END_GET
END_PROPERTY

METHOD reset : BOOL // Return TRUE if finish.
VAR_INPUT
	deep : BOOL := FALSE;
END_VAR
VAR
	_reset_children :BOOL := FALSE;
END_VAR
// Waiting finish process and remove jobs from container items.
IF THIS^.busy THEN
	THIS^.abort();
ELSIF _interface_container <> 0 AND _future <> 0 AND_THEN 
	( NOT _future.persistent_future OR deep) THEN
	_reset_children := _interface_container.reset(deep);
ELSE
	_reset_children := TRUE;
END_IF

// Remove my future.
IF _reset_children AND _future <> 0 THEN
	IF  NOT _future.persistent_future OR deep THEN
		IF _future_creator <> 0 THEN
			_future := _future_creator.destroy_future(_future);
		ELSIF _future.init() THEN
			_future.state := E_FutureExecutionState.idle;
			_future := 0;
		END_IF
		IF _future = 0 THEN
			_interface_container := 0;
			reset := TRUE;
		END_IF
	ELSE
		IF _future.init() THEN
			reset := TRUE;
		END_IF
	END_IF
END_IF
END_METHOD

METHOD resume : BOOL
VAR_INST
	_executor : REFERENCE TO FB_Executor;
END_VAR
_resume := TRUE;
IF _interface_container <> 0 THEN
	IF NOT _interface_container.resume() THEN
		_resume := FALSE;
	END_IF
END_IF
IF NOT _resume THEN
	_future.execute();
END_IF
resume := _resume;
END_METHOD

PROPERTY serial : ULINT
GET
serial := _serial;
END_GET
SET
_serial := serial;
END_SET
END_PROPERTY

METHOD start : BOOL
VAR
	_start_children :BOOL := FALSE;
END_VAR
// Start my future.
_start := _state = E_FutureExecutionState.wait_for_process;
start := TRUE;
END_METHOD

PROPERTY transition : BOOL
GET
transition := _transition;
END_GET
END_PROPERTY

PROPERTY upstream_aborting : BOOL
GET
upstream_aborting := _upstream_aborting;
END_GET
SET
_upstream_aborting := upstream_aborting;
END_SET
END_PROPERTY

END_FUNCTION_BLOCK

// ---- POUs/model/library/Observer/FB_JobEventLogStr.TcPOU
FUNCTION_BLOCK FB_JobEventLogStr IMPLEMENTS I_Observer

METHOD notify : BOOL
VAR_INPUT
	publisher	: I_Observable;
END_VAR
VAR_INST
	fb_timezone_info : FB_GetTimeZoneInformation := (bExecute := TRUE);
	text : T_MaxString;
END_VAR
VAR
	job_info : I_JobInfo;
	container : I_Container;
	num_of_jobs : UDINT;
END_VAR

IF NOT __QUERYINTERFACE(publisher, job_info) THEN
	RETURN;
END_IF

IF job_info.job.children <> 0 THEN
	num_of_jobs := job_info.job.children.num_of_jobs;
ELSE
	num_of_jobs := 0;
END_IF

IF job_info.job <> 0 THEN
	text := '';
	//fb_timezone_info();
	//text := FILETIME64_TO_ISO8601(fileTime := job_report.record_time, nBias := DINT_TO_INT(fb_timezone_info.tzInfo.bias), bUTC := TRUE,nPrecision := 6);
	//text := CONCAT(text, ' ');
	//text := CONCAT(text, job_report.title);
	text := CONCAT(text, '		');
	text := CONCAT(text, job_info.job.id);
	text := CONCAT(text, '		');
	text := CONCAT(text, job_info.job.namespace);
	text := CONCAT(text, '		');
	text := CONCAT(text, TO_STRING(num_of_jobs));
	text := CONCAT(text, '		');
	text := CONCAT(text, TO_STRING(job_info.new_state));
	text := CONCAT(text, '		');
	text := CONCAT(text, TO_STRING(job_info.job.nErrorID));
	text := CONCAT(text, '		');
	text := CONCAT(text, job_info.job.future.future_name);
	
	ADSLOGSTR(msgCtrlMask := ADSLOG_MSGTYPE_LOG,
 			 msgFmtStr := text, 
			strArg := '');	
END_IF

notify := TRUE;
END_METHOD

END_FUNCTION_BLOCK

// ---- POUs/model/library/Observer/FB_JobEventCyclicOutput.TcPOU
FUNCTION_BLOCK FB_JobEventCyclicOutput IMPLEMENTS I_Observer
VAR_OUTPUT
	event_message : ST_JobEventMessage;
END_VAR
VAR
	queue : FB_EventMessageQueue;
	cycle_counter : UINT;
END_VAR

IF queue.usage > 0 THEN
	event_message := queue.get();
END_IF

METHOD notify : BOOL
VAR_INPUT
	publisher	: I_Observable;
END_VAR
VAR_INST
	_event_message : ST_JobEventMessage;
END_VAR
VAR
	job_info : I_JobInfo;
	container : I_Container;
	num_of_jobs : UDINT;
END_VAR
IF NOT __QUERYINTERFACE(publisher, job_info) THEN
	RETURN;
END_IF

IF job_info.job.children <> 0 THEN
	num_of_jobs := job_info.job.children.num_of_jobs;
ELSE
	num_of_jobs := 0;
END_IF

_event_message.job_id := job_info.job.id;
_event_message.job_namespace := job_info.job.namespace;
_event_message.num_of_job := num_of_jobs;
_event_message.new_state := TO_STRING(job_info.new_state);
_event_message.old_state := TO_STRING(job_info.last_state);
_event_message.record_time := job_info.record_time;
_event_message.subject := job_info.job.future.future_name;
queue.put(_event_message);
notify := TRUE;
END_METHOD

END_FUNCTION_BLOCK

// ---- POUs/model/activities/FB_EventMessageQueue.TcPOU
FUNCTION_BLOCK FB_EventMessageQueue
VAR CONSTANT
	COMMAND_QUEUE_BUFFER_SIZE :UDINT := 50;
END_VAR
VAR_OUTPUT
END_VAR
VAR
	_usage:	UDINT;
	_write_index : UDINT := 1;
	_read_index : UDINT := 1;
	_queue_size:	UDINT := COMMAND_QUEUE_BUFFER_SIZE;
	queue_buffer:	ARRAY [1..COMMAND_QUEUE_BUFFER_SIZE] OF ST_JobEventMessage;
END_VAR

PROPERTY full : BOOL
GET
full :=  _usage >= COMMAND_QUEUE_BUFFER_SIZE;
END_GET
END_PROPERTY

METHOD get : REFERENCE TO ST_JobEventMessage
VAR_INPUT
END_VAR
IF _usage = 0 THEN
	get REF= 0;
	RETURN;
END_IF

get REF= queue_buffer[_read_index];

_usage := _usage - 1;

IF COMMAND_QUEUE_BUFFER_SIZE > _read_index THEN
	_read_index := _read_index + 1;
ELSE
	_read_index := 1;
END_IF
END_METHOD

METHOD put : BOOL
VAR_INPUT
	fbEvent:	REFERENCE TO ST_JobEventMessage;
END_VAR
IF _usage >= COMMAND_QUEUE_BUFFER_SIZE THEN
	put := FALSE;
ELSE
	queue_buffer[_write_index] := fbEvent;
	_usage := _usage + 1;
	IF COMMAND_QUEUE_BUFFER_SIZE > _write_index THEN
		_write_index := _write_index + 1;
	ELSE
		_write_index := 1;
	END_IF
	put := TRUE;
END_IF
END_METHOD

PROPERTY usage : UDINT
GET
usage := _usage;
END_GET
END_PROPERTY

END_FUNCTION_BLOCK

// ---- POUs/model/activities/FutureMCPower.TcPOU
{attribute 'enable_dynamic_creation'}
FUNCTION_BLOCK FutureMCPower EXTENDS FB_AbstructFuture
VAR_INPUT
END_VAR
VAR_OUTPUT
END_VAR
VAR
	_axis: REFERENCE TO AXIS_REF;
	_override: LREAL := 100.0;
	_enable_positive:	BOOL := TRUE; 
	_enable_negative:	BOOL := TRUE;
	_fb_power	: MC_Power;
	_mc_reset	: MC_Reset;
	_mc_stop	: MC_Stop;
	_option : ST_PowerOptions;
	_buffer_mode : MC_BufferMode;
	_status : BOOL;
END_VAR

METHOD error_reset : BOOL // Must be overrided if future has any errors.
VAR_INST
	_exec_state : UDINT;
END_VAR
IF _error_id <> 0 THEN
	CASE _exec_state OF
		0:
			_mc_reset(Axis := _axis, Execute := FALSE);
			_mc_reset(Axis:= _axis, Execute := TRUE );
			_exec_state := 1;
		1:
			IF _mc_reset.Busy THEN
				_mc_reset(Axis:= _axis,Execute := FALSE);
				error_reset := TRUE;
			END_IF
	END_CASE	
	_error_id := _fb_power.ErrorID;
ELSE
	error_reset := TRUE;
END_IF
END_METHOD

METHOD execute : BOOL // Return TRUE if finish.
VAR_INST
	_exec_state: UINT;
	_stoped : BOOL;
END_VAR
_axis.ReadStatus();
IF _axis.Status.Moving THEN
	_stoped := FALSE;
	_exec_state := 0;
END_IF

IF NOT _stoped THEN
	CASE _exec_state OF
		0:
			_mc_stop(axis := _axis, Execute := FALSE);
			_mc_stop(
				Axis:= _axis,
				Execute := TRUE
			);
			_exec_state := 1;
		1:
			IF _mc_stop.Busy THEN
				_mc_stop(Axis:= _axis,Execute := FALSE);
				_stoped := TRUE;
			END_IF
	END_CASE
END_IF
	
IF _axis.Status.NotMoving AND _stoped THEN
	_fb_power(
		Axis:= _axis, 
		Enable:= _status, 
		Enable_Positive:= _enable_positive, 
		Enable_Negative:= _enable_negative, 
		Override:= _override, 
		BufferMode:= _buffer_mode, 
		Options:= _option, 
	);
	_error_id := _fb_power.ErrorID;
	execute := _status = _fb_Power.Status;
END_IF
END_METHOD

METHOD set_options : BOOL
VAR_INPUT
	Enable_Positive:	BOOL; 
	Enable_Negative:	BOOL;
	Override:			LREAL := 100;
	buffer_mode : MC_BufferMode;
	option : ST_PowerOptions;
END_VAR
_override := Override;
_enable_positive := Enable_Positive;
_enable_negative := Enable_Negative;
_buffer_mode := buffer_mode;
_option := option;
END_METHOD

METHOD set_parameters : BOOL
VAR_INPUT
	axis : REFERENCE TO AXIS_REF;
	status : BOOL;
END_VAR
_axis REF= axis;
_status := status;
_enable_positive := status;
_enable_negative := status;
END_METHOD

END_FUNCTION_BLOCK

// ---- POUs/model/library/FB_AbstructFuture.TcPOU
FUNCTION_BLOCK ABSTRACT FB_AbstructFuture IMPLEMENTS I_Future
VAR_INPUT
END_VAR
VAR_OUTPUT
END_VAR
VAR
	_executor : I_Job;
	{attribute 'TcEncoding':='UTF-8'}
	_future_name :STRING := 'NO_NAME';
	_busy : BOOL; 
	_persistent_future : BOOL;
	_state : E_FutureExecutionState;
	_error_id : HRESULT;
END_VAR

METHOD abort : BOOL // Must be overrided if future has any errors.
abort := TRUE;
END_METHOD

METHOD error_reset : BOOL // Must be overrided if future has any errors.
error_reset := TRUE;
END_METHOD

METHOD execute : BOOL // Must be overrided.
END_METHOD

PROPERTY executor : I_Job
GET
executor := _executor;
END_GET
SET
_executor := executor;
END_SET
END_PROPERTY

PROPERTY future_name : STRING // Name of future.
GET
future_name := _future_name;
END_GET
SET
_future_name := future_name;
END_SET
END_PROPERTY

METHOD init : BOOL // Return TRUE if finish.
init := TRUE;
END_METHOD

PROPERTY nErrorID : HRESULT // Must be overrided if future has any errors.
GET
nErrorID := _error_id;
END_GET
END_PROPERTY

PROPERTY persistent_future : BOOL
GET
persistent_future := _persistent_future;
END_GET
SET
_persistent_future := persistent_future;
END_SET
END_PROPERTY

METHOD quit : BOOL // Return TRUE if finish.
init();
quit := TRUE;
END_METHOD

PROPERTY state : E_FutureExecutionState // Execution state of this future.
GET
state := _state;
END_GET
SET
_state := state;
END_SET
END_PROPERTY

END_FUNCTION_BLOCK

// ---- POUs/model/library/FB_BatchJobContainer.TcPOU
{attribute 'enable_dynamic_creation'}
FUNCTION_BLOCK FB_BatchJobContainer EXTENDS FB_AbstructContainer IMPLEMENTS I_SerialContainer
VAR_INPUT
END_VAR
VAR_OUTPUT
END_VAR
VAR
	_all_abort : BOOL;
	current_executing_future_id : UINT;
	current_executing_future : I_Future;
END_VAR

METHOD PROTECTED _append_job : BOOL
VAR_INPUT
	executor	: I_Job;
END_VAR
VAR
	_parent_future_id: STRING;	
END_VAR
IF executor <> 0 AND _num_of_jobs < ParamFuturesLib.MAX_TASK_NUM THEN
	executor.init();
	IF _num_of_jobs > 0 THEN
		_executors[_num_of_jobs].next_job := executor;
		executor.previous_job := _executors[_num_of_jobs];
	END_IF
	_num_of_jobs := _num_of_jobs + 1;
	executor.serial := TO_ULINT(_num_of_jobs);
	
	_executors[_num_of_jobs] := executor;
	IF  _executor <> 0 THEN
		// Propergate task creator object
		_executors[_num_of_jobs].job_event_observable := _executor.job_event_observable;
		_executors[_num_of_jobs].parent_executor := _executor;
		_executors[_num_of_jobs].upstream_aborting := _executor.upstream_aborting;
		_parent_future_id := _executor.id;
	END_IF
END_IF
END_METHOD

(* This is the generator that iteratively generates references to FB_executor instances*)
METHOD _index_generator_ : UINT
VAR_INST
	_index : UINT;
END_VAR
_index := _index + 1;
IF _index > _num_of_jobs THEN
	_index := 0;
END_IF
_index_generator_ := _index;
END_METHOD

METHOD abort : BOOL // Return TRUE if finish.
IF current_executing_future_id > 1 AND ParamFuturesLib.MAX_TASK_NUM <= current_executing_future_id THEN
	abort := _executors[current_executing_future_id].abort();
ELSE
	abort := TRUE;
END_IF
END_METHOD

PROPERTY current_job : I_Job
GET
current_job := _executors[current_executing_future_id];
END_GET
END_PROPERTY

METHOD execute : BOOL // Return TRUE if finish.
VAR_INST
	i :UDINT;
	complete_last_proess :BOOL;
	complete_all_process :BOOL;
END_VAR
IF _num_of_jobs = 0 THEN
	RETURN;
END_IF



FOR i := 1 TO _num_of_jobs DO
	complete_all_process := _executors[i].execute();
	_error_id := _executors[i].nErrorID;
END_FOR

IF current_executing_future_id > 1 THEN
	complete_last_proess := _executors[current_executing_future_id - 1].done;
ELSE
	complete_last_proess := TRUE;
END_IF

CASE _executors[current_executing_future_id].current_state OF
	E_FutureExecutionState.init, E_FutureExecutionState.process, E_FutureExecutionState.quit:
		_all_abort := FALSE;
		IF _abort THEN
			IF _executors[current_executing_future_id].abort() THEN
				_all_abort := TRUE;
			END_IF
		END_IF
	E_FutureExecutionState.wait_for_process:
		IF _executors[current_executing_future_id].ready AND complete_last_proess AND SUPER^._auto_start THEN
			_executors[current_executing_future_id].start();
		END_IF
END_CASE

IF complete_all_process THEN
	execute := NOT _continuous_mode;
ELSIF _executors[current_executing_future_id].done AND current_executing_future_id < _num_of_jobs THEN
	execute := FALSE;
	current_executing_future_id := current_executing_future_id + 1;
END_IF

current_executing_future := _executors[current_executing_future_id].future;
END_METHOD

METHOD init : BOOL // Return TRUE if finish.
VAR
	_executor : I_Job;
	_init_done : BOOL;
END_VAR
_init_done := TRUE;
REPEAT
	_executor := each_executor;
	IF _executor <> 0 THEN
		IF NOT _executor.init() THEN
			_init_done := FALSE;
		END_IF
	END_IF
UNTIL
	_executor = 0
END_REPEAT

current_executing_future_id := 1;
_error_id := 0;
init := _init_done;
END_METHOD

METHOD quit : BOOL // Return TRUE if finish.
VAR_INST
	i: UDINT;
	complete_all_task :BOOL;
END_VAR
complete_all_task := TRUE;
FOR i := 1 TO _num_of_jobs DO
	_executors[i].execute();
	IF NOT (_executors[i].current_state = E_FutureExecutionState.finish) THEN
		complete_all_task := FALSE;	
	END_IF
END_FOR
IF complete_all_task THEN
	current_executing_future_id := 1;
	quit := TRUE;
ELSE
	quit := FALSE;
END_IF
END_METHOD

METHOD resume : BOOL
IF current_executing_future_id > 1 AND ParamFuturesLib.MAX_TASK_NUM <= current_executing_future_id THEN
	resume := _executors[current_executing_future_id].resume();
ELSE
	resume := TRUE;
END_IF
END_METHOD

END_FUNCTION_BLOCK

// ---- POUs/model/library/FB_AbstructContainer.TcPOU
FUNCTION_BLOCK ABSTRACT FB_AbstructContainer EXTENDS FB_AbstructFuture IMPLEMENTS I_Container
VAR_INPUT
END_VAR
VAR_OUTPUT
END_VAR
VAR
	_executors : ARRAY [1..ParamFuturesLib.MAX_TASK_NUM] OF I_Job;
	_start :BOOL;
	_auto_start : BOOL := TRUE;
	_abort : BOOL;
	_num_of_jobs: UDINT;
	_continuous_mode : BOOL;
	_job_event_reporter : I_JobInfo;
	_serial_id : ULINT;
END_VAR

METHOD PROTECTED _append_job : BOOL
VAR_INPUT
	executor	: I_Job;
END_VAR
_serial_id := _serial_id + 1;
executor.serial := _serial_id;
END_METHOD

(* This is the generator that iteratively generates references to FB_executor instances*)
METHOD _index_generator_ : UINT
VAR_INST
	_index : UINT;
END_VAR
_index := _index + 1;
IF _index > _num_of_jobs THEN
	_index := 0;
END_IF
_index_generator_ := _index;
END_METHOD

METHOD abort : BOOL // Return TRUE if finish.
END_METHOD

METHOD append_job : I_Job
VAR_INPUT
	executor	: I_Job;
END_VAR
executor.persistent_job := TRUE;
THIS^._append_job(executor);
append_job := executor;
END_METHOD

{warning 'Add property implementation'}
PROPERTY auto_start : BOOL
GET
auto_start := _auto_start;
END_GET
SET
_auto_start := auto_start;
END_SET
END_PROPERTY

PROPERTY continuous_mode : BOOL
SET
VAR
	_executor : I_Job;
END_VAR
_continuous_mode := continuous_mode;
REPEAT
	_executor := THIS^.each_executor;
	IF _executor <> 0 THEN
		_executor.continuous_mode := continuous_mode;
	END_IF
UNTIL
	_executor = 0
END_REPEAT
END_SET
END_PROPERTY

METHOD create_container : I_Job
VAR_INPUT
	container_type	: ContainerType;
	name	: STRING;
END_VAR
CASE container_type OF
	ContainerType.BATCH:
		create_container := THIS^.create_job(GVL.batch_job_container_creator,name);
	ContainerType.PARALLEL:
		create_container := THIS^.create_job(GVL.parallel_job_container_creator,name);
	ContainerType.QUEUE:
		create_container := THIS^.create_job(GVL.queue_job_container_creator,name);
	ContainerType.PARALLEL_QUEUE:
		create_container := THIS^.create_job(GVL.parallel_queue_job_container_creator,name);
END_CASE
END_METHOD

METHOD create_job : I_Job
VAR_INPUT
	creator	: I_TaskCreator;
	future_name	: STRING;
END_VAR
VAR
	future : I_Future;
END_VAR
IF _num_of_jobs < ParamFuturesLib.MAX_TASK_NUM THEN
	future := creator.create_future(future_name);
	create_job := THIS^.spawn_job(future);
	create_job.persistent_job := FALSE;
	IF create_job <> 0 THEN
		create_job.future_creator := creator;
	ELSE
		creator.destroy_future(future);
	END_IF
END_IF
END_METHOD

PROPERTY each_executor : I_Job
GET
VAR
	_index : UINT;
END_VAR
_index := _index_generator_();
IF _index > 0 THEN
	IF _executors[_index] <> 0 THEN
		IF _executors[_index] <> 0 THEN
			each_executor := _executors[_index];
		ELSE
			each_executor := 0;
		END_IF
	END_IF
ELSE
	each_executor := 0;
END_IF
END_GET
END_PROPERTY

METHOD error_reset : BOOL
VAR
	_executor : I_Job;
	complete : BOOL;
END_VAR
complete := TRUE;
REPEAT
	_executor := each_executor;
	IF _executor <> 0 THEN
		IF NOT _executor.error_reset() THEN
			complete := FALSE;
		END_IF
	END_IF
UNTIL
	_executor = 0
END_REPEAT
IF complete THEN
	_error_id := 0;
END_IF
error_reset := complete;
END_METHOD

METHOD init : BOOL // Return TRUE if finish.
VAR
	_each_executor : i_Job;
	_init_done : BOOL;
END_VAR
_init_done := TRUE;
REPEAT
	_each_executor := THIS^.each_executor;
	IF _each_executor <> 0 THEN
		IF NOT _each_executor.init() THEN
			_init_done := FALSE;
		END_IF
	END_IF
UNTIL
	_each_executor = 0
END_REPEAT

_error_id := 0;
init := _init_done;
END_METHOD

PROPERTY num_of_jobs : UDINT
GET
num_of_jobs := _num_of_jobs;
END_GET
END_PROPERTY

METHOD reset : BOOL // Return TRUE if finish.
VAR_INPUT
	deep : BOOL := FALSE;
END_VAR
VAR
	i : UINT;
	_delete_counter : UINT;
	_p_executor : POINTER TO FB_Executor;
	text : STRING;
END_VAR
_delete_counter := 0;
REPEAT
	i := _index_generator_();
	IF _num_of_jobs > _delete_counter AND i > 0 THEN
		IF _executors[i] <> 0 THEN
			IF _executors[i].reset(deep) THEN
				IF __QUERYPOINTER(_executors[i],_p_executor) THEN
					__DELETE(_p_executor);
				ELSE
					_executors[i] := 0;
				END_IF
				_delete_counter := _delete_counter + 1;
			END_IF
		END_IF
	END_IF
UNTIL
	i = 0
END_REPEAT
_num_of_jobs := _num_of_jobs - _delete_counter;
reset := _num_of_jobs = 0;
END_METHOD

METHOD resume : BOOL
VAR
	_all_done : BOOL;
END_VAR
VAR_INST
	_executor : I_Job;
END_VAR
_all_done := TRUE;
REPEAT
	_executor := THIS^.each_executor;
	IF _executor <> 0 THEN
		IF NOT _executor.resume() THEN
			_all_done := FALSE;
		END_IF
	END_IF
UNTIL
	_executor = 0
END_REPEAT
resume := _all_done;
END_METHOD

METHOD spawn_job : I_Job
VAR_INPUT
	future : I_Future;
	job_persistence : BOOL := FALSE;
END_VAR
VAR
	_spawned_executor : POINTER TO FB_Executor;
END_VAR
IF future <> 0 THEN
	_spawned_executor := __NEW(FB_Executor);
	_spawned_executor^.future := future;
	_spawned_executor^.persistent_job := job_persistence;
	_append_job(_spawned_executor^);
	spawn_job := _spawned_executor^;
ELSE
	spawn_job := 0;
END_IF
END_METHOD

PROPERTY state : E_FutureExecutionState
GET
state := _state;
END_GET
SET
_state := state;
END_SET
END_PROPERTY

END_FUNCTION_BLOCK

// ---- POUs/model/activities/FutureSleep.TcPOU
{attribute 'enable_dynamic_creation'}
FUNCTION_BLOCK FutureSleep EXTENDS FB_AbstructFuture
VAR_INPUT
END_VAR
VAR_OUTPUT
END_VAR
VAR
	_sleep_timer : TON;
	_sleep_time: TIME;
END_VAR

METHOD execute : BOOL // Return TRUE if finish.
_sleep_timer(IN := TRUE, PT := _sleep_time);
execute := _sleep_timer.Q;
END_METHOD

METHOD init : BOOL // Return TRUE if finish.
_sleep_timer(IN := FALSE);
init := TRUE;
END_METHOD

PROPERTY sleep_time : TIME
GET
sleep_time := _sleep_timer.ET;
END_GET
SET
_sleep_time := sleep_time;
END_SET
END_PROPERTY

END_FUNCTION_BLOCK

// ---- POUs/model/activities/FutureSleepCreator.TcPOU
FUNCTION_BLOCK FutureSleepCreator IMPLEMENTS I_TaskCreator
VAR_INPUT
END_VAR
VAR_OUTPUT
END_VAR
VAR
	_sleep_time: TIME;
	_p_future : POINTER TO FutureSleep;
END_VAR

{warning 'add method implementation '}
METHOD create_future : I_Future
VAR_INPUT
	(* Specify future name*)
	future_name	: STRING;
END_VAR
_p_future := __NEW(FutureSleep);
_p_future^.future_name := future_name;
_p_future^.sleep_time := _sleep_time;
create_future := _p_future^;
END_METHOD

{warning 'add method implementation '}
METHOD destroy_future : I_Future
VAR_INPUT
	(* Specify future instance whtat you want to delete.*)
	future	: I_Future;
END_VAR
VAR
	_p_future : POINTER TO FutureSleep;
END_VAR
IF __QUERYPOINTER(future, _p_future) THEN
	__DELETE(_p_future);
	IF _p_future = 0  THEN
		destroy_future := 0;
	END_IF
END_IF
END_METHOD

PROPERTY sleep_time : TIME
GET
sleep_time := _p_future^.sleep_time;
END_GET
SET
_sleep_time := sleep_time;
END_SET
END_PROPERTY

END_FUNCTION_BLOCK

// ---- POUs/model/activities/FutureMCMoveRelativeCreator.TcPOU
FUNCTION_BLOCK FutureMCMoveRelativeCreator IMPLEMENTS I_TaskCreator
VAR_INPUT
END_VAR
VAR_OUTPUT
END_VAR
VAR
	_axis: REFERENCE TO AXIS_REF;
	_distance : MC_LREAL;
	_velocity : MC_LREAL;
	_acceleration: MC_LREAL;
	_deceleration: MC_LREAL;
	_jerk		: MC_LREAL;
	_option : ST_MoveOptions;
	_buffer_mode : MC_BufferMode ;
END_VAR

{warning 'add method implementation '}
METHOD create_future : I_Future
VAR_INPUT
	(* Specify future name*)
	future_name	: STRING;
END_VAR
VAR
	_p_future : POINTER TO FutureMCMoveRelative;
END_VAR
_p_future := __NEW(FutureMCMoveRelative);
_p_future^.future_name := future_name;
_p_future^.set_parameters(_axis, _distance, _velocity, _acceleration, _deceleration,_jerk ,_buffer_mode);
_p_future^.set_options( _option);
create_future := _p_future^;
END_METHOD

{warning 'add method implementation '}
METHOD destroy_future : I_Future
VAR_INPUT
	(* Specify future instance whtat you want to delete.*)
	future	: I_Future;
END_VAR
VAR
	_p_future : POINTER TO FutureMCMoveRelative;
END_VAR
IF __QUERYPOINTER(future, _p_future) THEN
	__DELETE(_p_future);
	IF _p_future = 0  THEN
		destroy_future := 0;
	END_IF
END_IF
END_METHOD

METHOD set_options : BOOL
VAR_INPUT
	option : ST_MoveOptions;
END_VAR
_option := option;
END_METHOD

METHOD set_parameters : BOOL
VAR_INPUT
	axis : REFERENCE TO AXIS_REF;
	distance : MC_LREAL;
	velocity : MC_LREAL;
	acceleration	: MC_LREAL;		// Set deceleration in case let moving axis halt.
	deceleration	: MC_LREAL;		// Set deceleration in case let moving axis halt.
	jerk			: MC_LREAL;		// Set jerk in case let moving axis halt.
	buffer_mode : MC_BufferMode;
END_VAR
_axis REF= axis;
_distance := distance;
_velocity := velocity;
_acceleration := acceleration;
_deceleration := deceleration;
_jerk := jerk;
_buffer_mode := buffer_mode;
END_METHOD

END_FUNCTION_BLOCK

// ---- POUs/model/activities/FutureMCMoveRelative.TcPOU
{attribute 'enable_dynamic_creation'}
FUNCTION_BLOCK FutureMCMoveRelative EXTENDS FB_AbstructFuture
VAR_INPUT
END_VAR
VAR_OUTPUT
END_VAR
VAR
	_fb_move_rel	: MC_MoveRelative;
	_mc_stop		: MC_Stop;
	_mc_reset	: MC_Reset;
	_abort_executor		: FB_Executor;
	_axis: REFERENCE TO AXIS_REF;
	_distance : MC_LREAL;
	_velocity : MC_LREAL;
	_acceleration: MC_LREAL;
	_deceleration: MC_LREAL;
	_jerk		: MC_LREAL;
	_option : ST_MoveOptions;
	_buffer_mode : MC_BufferMode ;
	_exec_state : UDINT;
	_abort_state : UINT;
END_VAR

METHOD abort : BOOL // Return TRUE if finish.
VAR_INST
	future_stop : FutureMcStop;
END_VAR
CASE _abort_state OF
	0:
		_mc_stop(axis := _axis, Execute := FALSE);
		_mc_stop(
			Axis:= _axis,
			Execute := TRUE,
			Jerk := _jerk,
			Options := _option
		);
		_abort_state := 1;
	1:
		IF _mc_stop.Busy THEN
			_mc_stop(Axis:= _axis,Execute := FALSE);
		END_IF
		IF _mc_stop.Done OR _mc_stop.Error THEN
			abort := TRUE;		
		END_IF
		_error_id := _mc_stop.ErrorID;
END_CASE
END_METHOD

METHOD error_reset : BOOL // Must be overrided if future has any errors.
IF _error_id <> 0 THEN
	CASE _exec_state OF
		0:
			_mc_reset(Axis := _axis, Execute := FALSE);
			_mc_reset(Axis:= _axis, Execute := TRUE );
			_exec_state := 1;
		1:
			IF _mc_reset.Busy THEN
				_mc_reset(Axis:= _axis,Execute := FALSE);
			END_IF
	END_CASE
	
	_error_id := _mc_reset.ErrorID;
	error_reset := _mc_reset.Done;
ELSE
	error_reset := TRUE;
END_IF
END_METHOD

METHOD execute : BOOL // Return TRUE if finish.

CASE _exec_state OF
	0:
		_abort_state := 0;
		_fb_move_rel(Axis := _axis,Execute := FALSE);
		_fb_move_rel(
			Execute := TRUE,
			Axis := _axis,
			Distance := _distance,
			Velocity := _velocity,
			Acceleration := _acceleration,
			Deceleration := _deceleration,
			Jerk := _jerk,
			BufferMode := _buffer_mode,
			Options := _option
		);
		_exec_state := 1;
	1:
		IF _fb_move_rel.Busy THEN
			_fb_move_rel(Axis := _axis,Execute := FALSE);
		END_IF
END_CASE

_error_id := _fb_move_rel.ErrorID;
execute := _fb_move_rel.Done OR _fb_move_rel.Error;
END_METHOD

METHOD init : BOOL // Return TRUE if finish.

VAR
	axis: INT;
END_VAR
_exec_state := 0;
_abort_state := 0;
_error_id := _fb_move_rel.ErrorID;
init := TRUE;
END_METHOD

METHOD set_options : BOOL
VAR_INPUT
	option : ST_MoveOptions;
END_VAR
_option := option;
END_METHOD

METHOD set_parameters : BOOL
VAR_INPUT
	axis : REFERENCE TO AXIS_REF;
	distance : MC_LREAL;
	velocity : MC_LREAL;
	acceleration	: MC_LREAL;		// Set deceleration in case let moving axis halt.
	deceleration	: MC_LREAL;		// Set deceleration in case let moving axis halt.
	jerk			: MC_LREAL;		// Set jerk in case let moving axis halt.
	buffer_mode : MC_BufferMode;
END_VAR
_axis REF= axis;
_distance := distance;
_velocity := velocity;
_acceleration := acceleration;
_deceleration := deceleration;
_jerk := jerk;
_buffer_mode := buffer_mode;
END_METHOD

END_FUNCTION_BLOCK

// ---- POUs/model/activities/FutureMCStop.TcPOU
{attribute 'enable_dynamic_creation'}
FUNCTION_BLOCK FutureMCStop EXTENDS FB_AbstructFuture
VAR_INPUT
END_VAR
VAR_OUTPUT
END_VAR
VAR
	_axis: REFERENCE TO AXIS_REF;
	_mc_stop	: MC_Stop;
	_mc_reset	: MC_Reset;
	_deceleration: MC_LREAL;
	_jerk		: MC_LREAL;
	_option : ST_MoveOptions;
	_exec_state : UDINT;
END_VAR

METHOD error_reset : BOOL // Must be overrided if future has any errors.
IF _error_id <> 0 THEN
	CASE _exec_state OF
		0:
			_mc_reset(Axis := _axis, Execute := FALSE);
			_mc_reset(Axis:= _axis, Execute := TRUE );
			_exec_state := 1;
		1:
			IF _mc_reset.Busy THEN
				_mc_reset(Axis:= _axis,Execute := FALSE);
			END_IF
	END_CASE
	
	_error_id := _mc_reset.ErrorID;
	error_reset := _mc_reset.Done;
ELSE
	error_reset := TRUE;
END_IF
END_METHOD

METHOD execute : BOOL // Return TRUE if finish.

CASE _exec_state OF
	0:
		_mc_stop(axis := _axis, Execute := FALSE);
		_mc_stop(
			Axis:= _axis,
			Execute := TRUE,
			Jerk := _jerk,
			Options := _option
		);
		_exec_state := 1;
	1:
		IF _mc_stop.Busy THEN
			_mc_stop(Axis:= _axis,Execute := FALSE);
		END_IF
END_CASE

_error_id := _mc_stop.ErrorID;
execute := _mc_stop.Done OR _mc_stop.Error;
END_METHOD

METHOD init : BOOL // Return TRUE if finish.
_exec_state := 0;
init := TRUE;
END_METHOD

METHOD set_options : BOOL
VAR_INPUT
	option : ST_MoveOptions;
END_VAR
_option := option;
END_METHOD

METHOD set_parameters : BOOL
VAR_INPUT
	axis : REFERENCE TO AXIS_REF;
	deceleration	: MC_LREAL;		// Set deceleration in case let moving axis halt.
	jerk			: MC_LREAL;		// Set jerk in case let moving axis halt.
END_VAR
_axis REF= axis;
_deceleration := deceleration;
_jerk := jerk;
END_METHOD

END_FUNCTION_BLOCK

// ---- POUs/model/activities/FutureMCMoveAbsoluteCreator.TcPOU
FUNCTION_BLOCK FutureMCMoveAbsoluteCreator IMPLEMENTS I_TaskCreator
VAR_INPUT
END_VAR
VAR_OUTPUT
END_VAR
VAR
	_axis: REFERENCE TO AXIS_REF;
	_position : MC_LREAL;
	_velocity : MC_LREAL;
	_acceleration: MC_LREAL;
	_deceleration: MC_LREAL;
	_jerk		: MC_LREAL;
	_option : ST_MoveOptions;
	_buffer_mode : MC_BufferMode ;
END_VAR

METHOD create_future : I_Future
VAR_INPUT
	(* Specify future name*)
	future_name	: STRING;
END_VAR
VAR
	_p_future : POINTER TO FutureMCMoveAbsolute;
END_VAR
_p_future := __NEW(FutureMCMoveAbsolute);
_p_future^.future_name := future_name;
_p_future^.set_parameters(_axis, _position, _velocity, _acceleration, _deceleration,_jerk ,_buffer_mode);
_p_future^.set_options( _option);
create_future := _p_future^;
END_METHOD

{warning 'add method implementation '}
METHOD destroy_future : I_Future
VAR_INPUT
	(* Specify future instance whtat you want to delete.*)
	future	: I_Future;
END_VAR
VAR
	_p_future : POINTER TO FutureMCMoveAbsolute;
END_VAR
IF __QUERYPOINTER(future, _p_future) THEN
	__DELETE(_p_future);
	IF _p_future = 0  THEN
		destroy_future := 0;
	END_IF
END_IF
END_METHOD

METHOD set_options : BOOL
VAR_INPUT
	option : ST_MoveOptions;
END_VAR
_option := option;
END_METHOD

METHOD set_parameters : BOOL
VAR_INPUT
	axis : REFERENCE TO AXIS_REF;
	position : MC_LREAL;
	velocity : MC_LREAL;
	acceleration	: MC_LREAL;		// Set deceleration in case let moving axis halt.
	deceleration	: MC_LREAL;		// Set deceleration in case let moving axis halt.
	jerk			: MC_LREAL;		// Set jerk in case let moving axis halt.
	buffer_mode : MC_BufferMode;
END_VAR
_axis REF= axis;
_position := position;
_velocity := velocity;
_acceleration := acceleration;
_deceleration := deceleration;
_jerk := jerk;
_buffer_mode := buffer_mode;
END_METHOD

END_FUNCTION_BLOCK

// ---- POUs/model/activities/FutureMCMoveAbsolute.TcPOU
{attribute 'enable_dynamic_creation'}
FUNCTION_BLOCK FutureMCMoveAbsolute EXTENDS FB_AbstructFuture
VAR_INPUT
END_VAR
VAR_OUTPUT
END_VAR
VAR
	_fb_move_abs	: MC_MoveAbsolute;
	_mc_stop		: MC_Stop;
	_mc_reset	: MC_Reset;
	_abort_executor		: FB_Executor;
	_axis: REFERENCE TO AXIS_REF;
	_position : MC_LREAL;
	_velocity : MC_LREAL;
	_acceleration: MC_LREAL;
	_deceleration: MC_LREAL;
	_jerk		: MC_LREAL;
	_option : ST_MoveOptions;
	_buffer_mode : MC_BufferMode ;
	_exec_state : UDINT;
	_abort_state : UINT;
END_VAR

METHOD abort : BOOL // Return TRUE if finish.
CASE _abort_state OF
	0:
		_mc_stop(axis := _axis, Execute := FALSE);
		_mc_stop(
			Axis:= _axis,
			Execute := TRUE,
			Jerk := _jerk,
			Options := _option
		);
		_abort_state := 1;
	1:
		IF _mc_stop.Busy THEN
			_mc_stop(Axis:= _axis,Execute := FALSE);
		END_IF
		IF _mc_stop.Done OR _mc_stop.Error THEN
			abort := TRUE;
		END_IF
		_error_id := _mc_stop.ErrorID;
END_CASE
END_METHOD

METHOD error_reset : BOOL // Must be overrided if future has any errors.
IF _error_id <> 0 THEN
	CASE _exec_state OF
		0:
			_mc_reset(Axis := _axis, Execute := FALSE);
			_mc_reset(Axis:= _axis, Execute := TRUE );
			_exec_state := 1;
		1:
			IF _mc_reset.Busy THEN
				_mc_reset(Axis:= _axis,Execute := FALSE);
			END_IF
	END_CASE
	
	_error_id := _mc_reset.ErrorID;
	error_reset := _mc_reset.Done;
ELSE
	error_reset := TRUE;
END_IF
END_METHOD

METHOD execute : BOOL // Return TRUE if finish.

CASE _exec_state OF
	0:
		_abort_state := 0;
		_fb_move_abs(Axis := _axis,Execute := FALSE);
		_fb_move_abs(
			Execute := TRUE,
			Axis := _axis,
			Position := _position,
			Velocity := _velocity,
			Acceleration := _acceleration,
			Deceleration := _deceleration,
			Jerk := _jerk,
			BufferMode := _buffer_mode,
			Options := _option
		);
		_exec_state := 1;
	1:
		IF _fb_move_abs.Busy THEN
			_fb_move_abs(Axis := _axis,Execute := FALSE);
		END_IF
END_CASE

_error_id := _fb_move_abs.ErrorID;
execute := _fb_move_abs.Done OR _fb_move_abs.Error;
END_METHOD

METHOD init : BOOL // Return TRUE if finish.
_exec_state := 0;
_abort_state := 0;
_error_id := _fb_move_abs.ErrorID;
init := TRUE;
END_METHOD

METHOD set_options : BOOL
VAR_INPUT
	option : ST_MoveOptions;
END_VAR
_option := option;
END_METHOD

METHOD set_parameters : BOOL
VAR_INPUT
	axis : REFERENCE TO AXIS_REF;
	position : MC_LREAL;
	velocity : MC_LREAL;
	acceleration	: MC_LREAL;		// Set deceleration in case let moving axis halt.
	deceleration	: MC_LREAL;		// Set deceleration in case let moving axis halt.
	jerk			: MC_LREAL;		// Set jerk in case let moving axis halt.
	buffer_mode : MC_BufferMode;
END_VAR
_axis REF= axis;
_position := position;
_velocity := velocity;
_acceleration := acceleration;
_deceleration := deceleration;
_jerk := jerk;
_buffer_mode := buffer_mode;
END_METHOD

END_FUNCTION_BLOCK

// ---- POUs/model/activities/FutureMCMoveVelocityCreator.TcPOU
FUNCTION_BLOCK FutureMCMoveVelocityCreator IMPLEMENTS I_TaskCreator
VAR_INPUT
END_VAR
VAR_OUTPUT
END_VAR
VAR
	_axis: REFERENCE TO AXIS_REF;
	_velocity : MC_LREAL;
	_direction : MC_DIRECTION;
	_acceleration: MC_LREAL;
	_deceleration: MC_LREAL;
	_jerk		: MC_LREAL;
	_option : ST_MoveOptions;
	_buffer_mode : MC_BufferMode ;
END_VAR

{warning 'add method implementation '}
METHOD create_future : I_Future
VAR_INPUT
	(* Specify future name*)
	future_name	: STRING;
END_VAR
VAR
	_p_future : POINTER TO FutureMCMoveVelocity;
END_VAR
_p_future := __NEW(FutureMCMoveVelocity);
_p_future^.future_name := future_name;
_p_future^.set_parameters(_axis, _direction, _velocity, _acceleration, _deceleration,_jerk ,_buffer_mode);
_p_future^.set_options( _option);
create_future := _p_future^;
END_METHOD

{warning 'add method implementation '}
METHOD destroy_future : I_Future
VAR_INPUT
	(* Specify future instance whtat you want to delete.*)
	future	: I_Future;
END_VAR
VAR
	_p_future : POINTER TO FutureMCMoveVelocity;
END_VAR
IF __QUERYPOINTER(future, _p_future) THEN
	__DELETE(_p_future);
	IF _p_future = 0  THEN
		destroy_future := 0;
	END_IF
END_IF
END_METHOD

METHOD set_options : BOOL
VAR_INPUT
	option : ST_MoveOptions;
END_VAR
_option := option;
END_METHOD

METHOD set_parameters : BOOL
VAR_INPUT
	axis : REFERENCE TO AXIS_REF;
	direction : MC_DIRECTION;
	velocity : MC_LREAL;
	acceleration	: MC_LREAL;		// Set deceleration in case let moving axis halt.
	deceleration	: MC_LREAL;		// Set deceleration in case let moving axis halt.
	jerk			: MC_LREAL;		// Set jerk in case let moving axis halt.
	buffer_mode : MC_BufferMode;
END_VAR
_axis REF= axis;
_velocity := velocity;
_direction := direction;
_acceleration := acceleration;
_deceleration := deceleration;
_jerk := jerk;
_buffer_mode := buffer_mode;
END_METHOD

END_FUNCTION_BLOCK

// ---- POUs/model/activities/FutureMCMoveVelocity.TcPOU
{attribute 'enable_dynamic_creation'}
FUNCTION_BLOCK FutureMCMoveVelocity EXTENDS FB_AbstructFuture
VAR_INPUT
END_VAR
VAR_OUTPUT
END_VAR
VAR
	_fb_move_velo	: MC_MoveVelocity;
	_mc_stop		: MC_Stop;
	_mc_reset	: MC_Reset;
	_abort_executor		: FB_Executor;
	_axis: REFERENCE TO AXIS_REF;
	_velocity : MC_LREAL;
	_direction : MC_DIRECTION;
	_acceleration: MC_LREAL;
	_deceleration: MC_LREAL;
	_jerk		: MC_LREAL;
	_option : ST_MoveOptions;
	_buffer_mode : MC_BufferMode ;
	_exec_state : UDINT;
	_abort_state : UINT;
END_VAR

METHOD abort : BOOL // Return TRUE if finish.
CASE _abort_state OF
	0:
		_mc_stop(axis := _axis, Execute := FALSE);
		_mc_stop(
			Axis:= _axis,
			Execute := TRUE,
			Jerk := _jerk,
			Options := _option
		);
		_abort_state := 1;
	1:
		IF _mc_stop.Busy THEN
			_mc_stop(Axis:= _axis,Execute := FALSE);
		END_IF
		IF _mc_stop.Done OR _mc_stop.Error THEN
			abort := TRUE;		
		END_IF
		_error_id := _mc_stop.ErrorID;
END_CASE
END_METHOD

METHOD error_reset : BOOL // Must be overrided if future has any errors.
IF _error_id <> 0 THEN
	CASE _exec_state OF
		0:
			_mc_reset(Axis := _axis, Execute := FALSE);
			_mc_reset(Axis:= _axis, Execute := TRUE );
			_exec_state := 1;
		1:
			IF _mc_reset.Busy THEN
				_mc_reset(Axis:= _axis,Execute := FALSE);
			END_IF
	END_CASE
	
	_error_id := _mc_reset.ErrorID;
	error_reset := _mc_reset.Done;
ELSE
	error_reset := TRUE;
END_IF
END_METHOD

METHOD execute : BOOL // Return TRUE if finish.

CASE _exec_state OF
	0:
		_abort_state := 0;
		_fb_move_velo(Axis := _axis,Execute := FALSE);
		_fb_move_velo(
			Execute := TRUE,
			Axis := _axis,
			Direction := _direction,
			Velocity := _velocity,
			Acceleration := _acceleration,
			Deceleration := _deceleration,
			Jerk := _jerk,
			BufferMode := _buffer_mode,
			Options := _option
		);
		_exec_state := 1;
	1:
		IF _fb_move_velo.Busy THEN
			_fb_move_velo(Axis := _axis,Execute := FALSE);
		END_IF
END_CASE

_error_id := _fb_move_velo.ErrorID;
execute := _fb_move_velo.InVelocity OR _fb_move_velo.Error;
END_METHOD

METHOD init : BOOL // Return TRUE if finish.

VAR
	axis: INT;
END_VAR
_exec_state := 0;
_abort_state := 0;
_error_id := _fb_move_velo.ErrorID;
init := TRUE;
END_METHOD

METHOD set_options : BOOL
VAR_INPUT
	option : ST_MoveOptions;
END_VAR
_option := option;
END_METHOD

METHOD set_parameters : BOOL
VAR_INPUT
	axis : REFERENCE TO AXIS_REF;
	direction : MC_DIRECTION;
	velocity : MC_LREAL;
	acceleration	: MC_LREAL;		// Set deceleration in case let moving axis halt.
	deceleration	: MC_LREAL;		// Set deceleration in case let moving axis halt.
	jerk			: MC_LREAL;		// Set jerk in case let moving axis halt.
	buffer_mode : MC_BufferMode;
END_VAR
_axis REF= axis;
_velocity := velocity;
_direction := direction;
_acceleration := acceleration;
_deceleration := deceleration;
_jerk := jerk;
_buffer_mode := buffer_mode;
END_METHOD

END_FUNCTION_BLOCK

// ---- POUs/model/activities/FutureMCStopCreator.TcPOU
FUNCTION_BLOCK FutureMCStopCreator IMPLEMENTS I_TaskCreator
VAR_INPUT
END_VAR
VAR_OUTPUT
END_VAR
VAR
	_axis: REFERENCE TO AXIS_REF;
	_deceleration: MC_LREAL;
	_jerk		: MC_LREAL;
	_option : ST_MoveOptions;
	_buffer_mode : MC_BufferMode;
END_VAR

{warning 'add method implementation '}
METHOD create_future : I_Future
VAR_INPUT
	(* Specify future name*)
	future_name	: STRING;
END_VAR
VAR
	_p_future : POINTER TO FutureMCStop;
END_VAR
_p_future := __NEW(FutureMCStop);
_p_future^.future_name := future_name;
_p_future^.set_parameters(_axis, _deceleration, _jerk);
_p_future^.set_options(_option);
create_future := _p_future^;
END_METHOD

{warning 'add method implementation '}
METHOD destroy_future : I_Future
VAR_INPUT
	(* Specify future instance whtat you want to delete.*)
	future	: I_Future;
END_VAR
VAR
	_p_future : POINTER TO FutureMCStop;
END_VAR
IF __QUERYPOINTER(future, _p_future) THEN
	__DELETE(_p_future);
	IF _p_future = 0  THEN
		destroy_future := 0;
	END_IF
END_IF
END_METHOD

METHOD set_options : BOOL
VAR_INPUT
	option : ST_MoveOptions;
END_VAR
_option := option;
END_METHOD

METHOD set_parameters : BOOL
VAR_INPUT
	axis : REFERENCE TO AXIS_REF;
	deceleration	: MC_LREAL;		// Set deceleration in case let moving axis halt.
	jerk			: MC_LREAL;		// Set jerk in case let moving axis halt.
END_VAR
_axis REF= axis;
_deceleration := deceleration;
_jerk := jerk;
END_METHOD

END_FUNCTION_BLOCK

// ---- POUs/model/library/FB_BatchJobContainerCreator.TcPOU
FUNCTION_BLOCK FB_BatchJobContainerCreator IMPLEMENTS I_TaskCreator
VAR_INPUT
END_VAR
VAR_OUTPUT
END_VAR
VAR
END_VAR

METHOD create_future : I_Future
VAR_INPUT
	future_name :STRING;
END_VAR
VAR
	_p_future : POINTER TO FB_BatchJobContainer;
END_VAR
_p_future := __NEW(FB_BatchJobContainer);
_p_future^.future_name := future_name;
create_future := _p_future^;
END_METHOD

{warning 'add method implementation '}
METHOD destroy_future : I_Future
VAR_INPUT
	future	: I_Future;
END_VAR
VAR
	_p_future : POINTER TO FB_BatchJobContainer;
END_VAR
IF __QUERYPOINTER(future, _p_future) THEN
	__DELETE(_p_future);
	IF _p_future = 0  THEN
		destroy_future := 0;
	END_IF
END_IF
END_METHOD

END_FUNCTION_BLOCK

// ---- POUs/model/library/FB_ParallelJobContainerCreator.TcPOU
FUNCTION_BLOCK FB_ParallelJobContainerCreator IMPLEMENTS I_TaskCreator
VAR_INPUT
END_VAR
VAR_OUTPUT
END_VAR
VAR
END_VAR

METHOD create_future : I_Future
VAR_INPUT
	future_name	: STRING;
END_VAR
VAR
	_p_future : POINTER TO FB_ParallelJobContainer;
END_VAR
_p_future := __NEW(FB_ParallelJobContainer);
_p_future^.future_name := future_name;
create_future := _p_future^;
END_METHOD

METHOD destroy_future : I_Future
VAR_INPUT
	future	: I_Future;
END_VAR
VAR
	_p_future : POINTER TO FB_ParallelJobContainer;
END_VAR
IF __QUERYPOINTER(future, _p_future) THEN
	__DELETE(_p_future);
	IF _p_future = 0  THEN
		destroy_future := 0;
	END_IF
END_IF
END_METHOD

END_FUNCTION_BLOCK

// ---- POUs/model/library/FB_ParallelJobContainer.TcPOU
{attribute 'enable_dynamic_creation'}
FUNCTION_BLOCK FB_ParallelJobContainer EXTENDS FB_AbstructContainer
VAR_INPUT
END_VAR
VAR_OUTPUT
END_VAR
VAR
	_initialize :BOOL;
END_VAR

METHOD PROTECTED _append_job : BOOL
VAR_INPUT
	executor	: I_Job;
END_VAR
VAR
	_parent_future_id :STRING;
END_VAR
IF executor <> 0 AND _num_of_jobs < ParamFuturesLib.MAX_TASK_NUM THEN
	executor.init();
	_num_of_jobs := _num_of_jobs + 1;
	executor.serial := TO_ULINT(_num_of_jobs);
	
	_executors[_num_of_jobs] := executor;
	IF  _executor <> 0 THEN
		// Propergate task creator object
		_executors[_num_of_jobs].job_event_observable := _executor.job_event_observable;
		_executors[_num_of_jobs].parent_executor := _executor;
		_executors[_num_of_jobs].upstream_aborting := _executor.upstream_aborting;
		_parent_future_id := _executor.id;
	END_IF
END_IF
END_METHOD

(* This is the generator that iteratively generates references to FB_executor instances*)
METHOD _index_generator_ : UINT
VAR_INST
	_index : UINT;
END_VAR
IF _index > _num_of_jobs THEN
	_index := 0;
ELSE
	_index := _index + 1;
END_IF
_index_generator_ := _index;
END_METHOD

METHOD abort : BOOL // Return TRUE if finish.
VAR
	_all_done : BOOL;
END_VAR
VAR_INST
	_executor : I_Job;
	await : BOOL;
END_VAR
_all_done := TRUE;
REPEAT
	_executor := each_executor;
	IF _executor <> 0 THEN
		await := _executor.abort();
		IF _executor.busy OR NOT await THEN
			_all_done := FALSE;			
		END_IF
	END_IF
UNTIL
	_executor = 0
END_REPEAT
abort := _all_done;
END_METHOD

METHOD execute : BOOL // Return TRUE if finish.
VAR_INST
	i :UDINT;
	complete_all_task :BOOL;
	wait_for_initilize :BOOL;
END_VAR
IF _num_of_jobs = 0 THEN
	RETURN;
END_IF

complete_all_task := TRUE;
FOR i := 1 TO _num_of_jobs DO
	// Execute all methods
	IF _executors[i].current_state < E_FutureExecutionState.finish THEN
		IF NOT _executors[i].execute() THEN
			complete_all_task := FALSE;
		END_IF
	END_IF
	
	CASE _executors[i].current_state OF 
		E_FutureExecutionState.wait_for_process:
			IF _executors[i].ready AND SUPER^._auto_start THEN
				_executors[i].start();
			END_IF
	END_CASE

	_error_id := 0;	
	IF FAILED(_executors[i].nErrorID) THEN
		_error_id := _executors[i].nErrorID;
	END_IF
END_FOR

execute := complete_all_task;
END_METHOD

METHOD init : BOOL // Return TRUE if finish.
VAR
	_executor : I_Job;
	_init_done : BOOL;
END_VAR
_init_done := TRUE;
REPEAT
	_executor := each_executor;
	IF _executor <> 0 THEN
		IF NOT _executor.init() THEN
			_init_done := FALSE;
		END_IF
	END_IF
UNTIL
	_executor = 0
END_REPEAT

_error_id := 0;
init := _init_done;
END_METHOD

METHOD quit : BOOL // Return TRUE if finish.
VAR_INST
	i: UDINT;
	complete_all_task :BOOL;
END_VAR
complete_all_task := TRUE;
FOR i := 1 TO _num_of_jobs DO
	IF NOT FAILED(_executors[i].nErrorID) THEN
		_executors[i].execute();
	ELSE
		_error_id := _executors[i].nErrorID;
	END_IF
	IF NOT (_executors[i].current_state = E_FutureExecutionState.finish) THEN
		complete_all_task := FALSE;	
	END_IF
END_FOR

IF complete_all_task THEN
	_initialize := FALSE;
	quit := TRUE;	
END_IF
END_METHOD

END_FUNCTION_BLOCK

// ---- POUs/model/library/FB_QueueJobContainerCreator.TcPOU
FUNCTION_BLOCK FB_QueueJobContainerCreator IMPLEMENTS I_TaskCreator
VAR_INPUT
END_VAR
VAR_OUTPUT
END_VAR
VAR
END_VAR

METHOD create_future : I_Future
VAR_INPUT
	future_name	: STRING;
END_VAR
VAR
	_p_future : POINTER TO FB_QueueJobContainer;
END_VAR
_p_future := __NEW(FB_QueueJobContainer);
_p_future^.future_name := future_name;
create_future := _p_future^;
END_METHOD

METHOD destroy_future : I_Future
VAR_INPUT
	future	: I_Future;
END_VAR
VAR
	_p_future : POINTER TO FB_QueueJobContainer;
END_VAR
IF __QUERYPOINTER(future, _p_future) THEN
	__DELETE(_p_future);
	IF _p_future = 0  THEN
		destroy_future := 0;
	END_IF
END_IF
END_METHOD

END_FUNCTION_BLOCK

// ---- POUs/model/library/FB_QueueJobContainer.TcPOU
{attribute 'enable_dynamic_creation'}
FUNCTION_BLOCK FB_QueueJobContainer EXTENDS FB_AbstructContainer IMPLEMENTS I_SerialContainer
VAR_INPUT
END_VAR
VAR_OUTPUT
END_VAR
VAR
	_current_executing_job : I_Job;
	nWriteIndex: 	UINT := 1;
	nReadIndex: 	UINT := 1;
END_VAR

METHOD PROTECTED _append_job : BOOL
VAR_INPUT
	executor	: I_Job;
END_VAR
VAR_INST
	carry_flag	: BOOL;
	last_index	: UINT := 1;
END_VAR
VAR
	_p_executor : POINTER TO FB_Executor;
END_VAR

//Set buffer index
IF executor <> 0 AND _num_of_jobs < ParamFuturesLib.MAX_TASK_NUM THEN
	IF _executors[nWriteIndex] <> 0 AND_THEN NOT _executors[nWriteIndex].persistent_job AND __QUERYPOINTER(_executors[nWriteIndex], _p_executor) THEN
		__DELETE(_p_executor);
	END_IF
	// Spawn new task with specified feature
	_executors[nWriteIndex] := executor;

	// Get parent tssk id
	IF _executor <> 0 THEN
		_executors[nWriteIndex].job_event_observable := _executor.job_event_observable;
		_executors[nWriteIndex].parent_executor := _executor;
		_executors[nWriteIndex].upstream_aborting := _executor.upstream_aborting;
	END_IF

	// Add reference to next, previous jobs 
	IF _executors[last_index] <> 0 THEN
		_executors[last_index].next_job := _executors[nWriteIndex];
		_executors[nWriteIndex].previous_job := _executors[last_index];
	END_IF

	last_index := nWriteIndex;


	// Prepare index for next added job
	nWriteIndex := _get_next_index(nWriteIndex);
	
	// Clear previous job pointer of prepared next job.
	IF _executors[nWriteIndex] <> 0 THEN
		_executors[nWriteIndex].previous_job := 0;
	END_IF

	// calculate number of jobs by queue address
	IF nWriteIndex = nReadIndex AND _num_of_jobs = ParamFuturesLib.MAX_TASK_NUM - 1 THEN 
		carry_flag := TRUE;
	END_IF

	IF carry_flag THEN
		_num_of_jobs := ParamFuturesLib.MAX_TASK_NUM;
		carry_flag := FALSE;
	ELSIF nWriteIndex >= nReadIndex THEN
		_num_of_jobs := nWriteIndex - nReadIndex;
	ELSE
		_num_of_jobs := ParamFuturesLib.MAX_TASK_NUM - nReadIndex + nWriteIndex;
	END_IF
	executor.init();


END_IF

SUPER^._append_job(executor);
END_METHOD

METHOD _get_next_index : UINT
VAR_INPUT
	cuurent_index : UINT;
END_VAR
_get_next_index := cuurent_index + 1;
IF _get_next_index > ParamFuturesLib.MAX_TASK_NUM THEN
	_get_next_index := 1;
END_IF
END_METHOD

(* This is the generator that iteratively generates references to FB_executor instances*)
METHOD _index_generator_ : UINT;
VAR_INST
	_init	: BOOL := FALSE;
	_index :UINT;
	_current_order_number : DINT;
	_carry_flag : BOOL;
END_VAR
IF NOT _init THEN
	_carry_flag := FALSE;
	_index := nReadIndex;
	_init := TRUE;
END_IF

// calculate order number of executing futures by queue address
IF _num_of_jobs = 0 THEN
	_current_order_number := 0;
ELSIF _carry_flag THEN // 
	_current_order_number := ParamFuturesLib.MAX_TASK_NUM;
ELSIF nWriteIndex > nReadIndex THEN // Normal case
	_current_order_number := _index - nReadIndex + 1;
ELSE // 
	_current_order_number := _index - nReadIndex + 1;
	IF _current_order_number < 0 THEN
		_current_order_number := _current_order_number + ParamFuturesLib.MAX_TASK_NUM;
	END_IF
	IF _current_order_number = ParamFuturesLib.MAX_TASK_NUM - 1 THEN
		_carry_flag := TRUE;
	END_IF
END_IF


_index_generator_ := _index;

//Set buffer index
IF _num_of_jobs = 0 OR _num_of_jobs < _current_order_number THEN
	_init := FALSE;
END_IF

IF NOT _init THEN
	_index_generator_ := 0;
END_IF

IF _init THEN
	_index := _index + 1;
	IF _index > ParamFuturesLib.MAX_TASK_NUM THEN
		_index := 1;
	END_IF
END_IF
END_METHOD

METHOD abort : BOOL // Return TRUE if finish.
VAR_INST
	await : BOOL;
END_VAR
IF _current_executing_job <> 0 THEN
	await := _current_executing_job.abort();
	abort := await AND NOT _current_executing_job.busy;
ELSE
	abort := TRUE;
END_IF
END_METHOD

PROPERTY current_job : I_Job
GET
current_job := _current_executing_job;
END_GET
END_PROPERTY

METHOD dequeue : I_Job;
VAR_INPUT
END_VAR
//Set buffer index
IF _num_of_jobs > 0 THEN
	dequeue := _executors[nReadIndex];
	nReadIndex := nReadIndex + 1;
	IF nReadIndex > ParamFuturesLib.MAX_TASK_NUM THEN
		nReadIndex := 1;
	END_IF
	// calculate order number of executing futures by queue address
	IF nWriteIndex >= nReadIndex THEN
		_num_of_jobs := nWriteIndex - nReadIndex;
	ELSE
		_num_of_jobs := ParamFuturesLib.MAX_TASK_NUM - nReadIndex + nWriteIndex;
	END_IF
ELSE
	dequeue := 0;
END_IF
END_METHOD

METHOD execute : BOOL // Return TRUE if finish.
VAR
	_head : BOOL;
	_execution_complete :BOOL; 
	_future_id :UINT;
	complete_last_proess :BOOL := FALSE;
	i: UINT;
	_finish_delay : TON;
	_executor : I_Job;

END_VAR
complete_last_proess := FALSE;

//IF _total_futures = 0 THEN
//	RETURN;
//END_IF

_head := TRUE;
REPEAT
	// キューインされたFB_executorインスタンスを順に取り出すイテレータ。_endがTRUEになれば全て取り出し完了。_headは先頭のみtrueになる。
	i := THIS^._index_generator_();
	
	IF i > 0 THEN
		_executor := _executors[i];
		_execution_complete := _executor.execute();
		
		CASE _executor.current_state OF
			E_FutureExecutionState.idle:
				_executor.init();
			E_FutureExecutionState.wait_for_process:
				IF _executor.ready AND (complete_last_proess OR _head) AND SUPER^._auto_start THEN
					_executor.start();
					_current_executing_job := _executor;
				END_IF
		END_CASE
		
		complete_last_proess := _executor.done;	

		_error_id := _executor.nErrorID;
		
		IF _execution_complete THEN
			IF _head THEN
				// キューの先頭がfinish状態になれば取り出してキューから削除する
				//IF _executor.reset(FALSE) THEN
					THIS^.dequeue();
				//END_IF
			END_IF		
		END_IF
	ELSIF  _execution_complete THEN
		execute := NOT _continuous_mode;
	END_IF
	_head := FALSE;
UNTIL
	i = 0
END_REPEAT;
END_METHOD

METHOD init : BOOL // Return TRUE if finish.
VAR
	_executor : I_Job;
	_init_done : BOOL;
END_VAR
_init_done := TRUE;
REPEAT
	_executor := each_executor;
	IF _executor <> 0 THEN
		IF NOT _executor.init() THEN
			_init_done := FALSE;
		END_IF
	END_IF
UNTIL
	_executor = 0
END_REPEAT

_current_executing_job := 0;
_error_id := 0;
init := _init_done;
END_METHOD

END_FUNCTION_BLOCK

// ---- POUs/model/library/FB_ParallelQueueJobContainerCreator.TcPOU
FUNCTION_BLOCK FB_ParallelQueueJobContainerCreator IMPLEMENTS I_TaskCreator
VAR_INPUT
END_VAR
VAR_OUTPUT
END_VAR
VAR
END_VAR

METHOD create_future : I_Future
VAR_INPUT
	future_name	: STRING;
END_VAR
VAR
	_p_future : POINTER TO FB_ParallelQueueJobContainer;
END_VAR
_p_future := __NEW(FB_ParallelQueueJobContainer);
_p_future^.future_name := future_name;
create_future := _p_future^;
END_METHOD

METHOD destroy_future : I_Future
VAR_INPUT
	future	: I_Future;
END_VAR
VAR
	_p_future : POINTER TO FB_ParallelQueueJobContainer;
END_VAR
IF __QUERYPOINTER(future, _p_future) THEN
	__DELETE(_p_future);
	IF _p_future = 0  THEN
		destroy_future := 0;
	END_IF
END_IF
END_METHOD

END_FUNCTION_BLOCK

// ---- POUs/model/library/FB_ParallelQueueJobContainer.TcPOU
{attribute 'enable_dynamic_creation'}
FUNCTION_BLOCK FB_ParallelQueueJobContainer EXTENDS FB_AbstructContainer
VAR_INPUT
END_VAR
VAR_OUTPUT
END_VAR

METHOD PROTECTED _append_job : BOOL
VAR_INPUT
	executor	: I_Job;
END_VAR
VAR
	_deteremine_index :  BOOL;
	_p_executor : POINTER TO FB_Executor;
	future_order_number: INT;
	_parent_future_id: STRING;
	i: 	UDINT := 1;
END_VAR
VAR_INST
	next_index : UDINT := 1;
	last_index : UDINT;
END_VAR
//Set buffer index
IF _num_of_jobs < ParamFuturesLib.MAX_TASK_NUM THEN
	i := next_index;
	_deteremine_index := FALSE;
	REPEAT
		IF i > ParamFuturesLib.MAX_TASK_NUM THEN
			_error_id := -8;
			RETURN;
		ELSIF _executors[i] = 0 THEN
			_deteremine_index := TRUE;
		ELSIF _executors[i].current_state <> E_FutureExecutionState.idle OR
			_executors[i].current_state <> E_FutureExecutionState.finish THEN
			IF NOT _executors[i].persistent_job AND __QUERYPOINTER(_executors[i], _p_executor) THEN
				__DELETE(_p_executor);
			END_IF
			_deteremine_index := TRUE;
		END_IF
		
		IF next_index >= ParamFuturesLib.MAX_TASK_NUM THEN
			next_index := 1;
		ELSE
			next_index := next_index + 1;
		END_IF
		IF NOT _deteremine_index THEN
			i := next_index;
		END_IF
		
	UNTIL
		_deteremine_index
	END_REPEAT

	// Spawn new task with specified future
	_executors[i] := executor;
	
	// Get parent task id
	IF _executor <> 0 THEN
		_executors[i].job_event_observable := _executor.job_event_observable;
		_executors[i].parent_executor := _executor;
		_executors[i].upstream_aborting := _executor.upstream_aborting;
		_parent_future_id := _executor.id;
	END_IF
	
	IF last_index > 0 AND_THEN _executors[last_index] <> 0 THEN
		_executors[last_index].next_job := _executors[i];
		_executors[i].previous_job := _executors[last_index];
	END_IF
	
	last_index := i;
	executor.init();
	
	_num_of_jobs := _num_of_jobs + 1;
END_IF

SUPER^._append_job(executor);
END_METHOD

(* This is the generator that iteratively generates references to FB_executor instances*)
METHOD _index_generator_ : UINT;
VAR_INPUT
END_VAR
VAR_INST
	_init	: BOOL := FALSE;
	_current_order_number : UINT; // Represent order number of iteration
	_index: UINT;
	_deteremine_index : BOOL;
END_VAR
IF NOT _init THEN
	_current_order_number := 0;
	_index := 1;
	_index_generator_ := 0;
	_init := TRUE;
END_IF

IF _num_of_jobs = 0 THEN
	RETURN;
END_IF


IF _current_order_number >= _num_of_jobs OR _index > ParamFuturesLib.MAX_TASK_NUM THEN
	_init := FALSE;
END_IF

IF _init THEN

	_deteremine_index := FALSE;
	REPEAT
		IF _index > ParamFuturesLib.MAX_TASK_NUM THEN
			_index_generator_ := 0;
			RETURN;
		ELSIF _executors[_index] = 0 THEN
			_index := _index + 1;
		ELSIF _executors[_index].current_state = E_FutureExecutionState.finish THEN
			IF _executors[_index].transition THEN
				_num_of_jobs := _num_of_jobs - 1;
				_deteremine_index := TRUE;
			ELSE
				_index := _index + 1;
			END_IF
		ELSE
			_deteremine_index := TRUE;
		END_IF
	UNTIL
		_deteremine_index
	END_REPEAT

	IF _executors[_index] <> 0 THEN
		_index_generator_ := _index;
	ELSE
		_index_generator_ := 0;
	END_IF
	_current_order_number := _current_order_number + 1;
	_index := _index + 1;
ELSE
	_index_generator_ := 0;
END_IF
END_METHOD

METHOD abort : BOOL // Return TRUE if finish.
VAR
	_all_done : BOOL;
END_VAR
VAR_INST
	_executor : I_Job;
	await : BOOL;
END_VAR
_all_done := TRUE;
REPEAT
	_executor := each_executor;
	IF _executor <> 0 THEN
		await := _executor.abort();
		IF _executor.busy OR NOT await THEN
			_all_done := FALSE;
		END_IF
	END_IF
UNTIL
	_executor = 0
END_REPEAT
abort := _all_done;
END_METHOD

METHOD execute : BOOL // Return TRUE if finish.
VAR
	_head : BOOL;
	_future_id :UINT;
	i: UINT;
END_VAR
execute := FALSE;

IF _num_of_jobs = 0 THEN
	RETURN;
END_IF

REPEAT
	// キューインされたFB_executorインスタンスを順に取り出すイテレータ。_endがTRUEになれば全て取り出し完了。_headは先頭のみtrueになる。
	i := _index_generator_();
	IF i > 0 THEN
		IF _executors[i].execute() THEN
			_executors[i].reset(FALSE);
			execute := _num_of_jobs = 0 AND NOT _continuous_mode;
		ELSE
			CASE _executors[i].current_state OF
				E_FutureExecutionState.idle:
					_executors[i].init();
				E_FutureExecutionState.wait_for_process:
					IF _executor.ready AND SUPER^._auto_start THEN
						_executors[i].start();
					END_IF
	
				//E_FutureExecutionState.init, E_FutureExecutionState.process, E_FutureExecutionState.quit:
				//	IF 	_executors[i].current_state = E_FutureExecutionState.process THEN
				//		// Report total futures
				//		current_executing_future := _executors[i].future;						
				//	END_IF
			END_CASE
			_error_id := _executors[i].nErrorID;
		END_IF
	END_IF
UNTIL
	i = 0
END_REPEAT
END_METHOD

METHOD init : BOOL // Return TRUE if finish.
VAR
	_executor : I_Job;
	_init_done : BOOL;
END_VAR
_init_done := TRUE;
REPEAT
	_executor := each_executor;
	IF _executor <> 0 THEN
		IF NOT _executor.init() THEN
			_init_done := FALSE;
		END_IF
	END_IF
UNTIL
	_executor = 0
END_REPEAT

_error_id := 0;
init := _init_done;
END_METHOD

END_FUNCTION_BLOCK

// ---- POUs/demo1.TcPOU
PROGRAM demo1
VAR
    init        : BOOL;
    demo_job    : FB_Executor;
    recipro_moving  : ARRAY [1..10] OF FutureMCMoveAbsolute;
	i : UDINT;
	
	state : UDINT;
	fb_power : MC_Power;
	runner : FB_TaskRunner;
	
END_VAR


IF NOT init THEN
    demo_job.create_container(ContainerType.BATCH, 'DEMO_JOB');
    FOR i := 1 TO 10 DO
        IF i mod 2 > 0 THEN
            recipro_moving[i].set_parameters(GVL.axis1,250,200,0,0,0,0);
			recipro_moving[i].future_name := 'Move +250 deg, 200 deg/s';
        ELSE
            recipro_moving[i].set_parameters(GVL.axis1,-250,200,0,0,0,0);
			recipro_moving[i].future_name := 'Move -250 deg, 200 deg/s';
        END_IF
        demo_job.children.spawn_job(recipro_moving[i]);        
    END_FOR
    init := TRUE;
END_IF


CASE state OF
	0:
		fb_power(
			Axis:= GVL.axis1, 
			Enable:= TRUE, 
			Enable_Positive:= TRUE, 
			Enable_Negative:= TRUE, 
			Override:= 100 
		);
		IF fb_power.Status = TRUE THEN
			state := 1;
		END_IF
	1:
		runner.append_job(demo_job);
		state := 2;
	2:
		IF demo_job.ready THEN
			demo_job.start();
		END_IF
		IF demo_job.done THEN
			state := 3;
		END_IF
	3:
		fb_power(
			Axis:= GVL.axis1, 
			Enable:= FALSE, 
			Enable_Positive:= FALSE, 
			Enable_Negative:= FALSE, 
			Override:= 100 
		);
END_CASE

runner();

END_PROGRAM

// ---- POUs/demo2.TcPOU
PROGRAM demo2
VAR
    init        : BOOL;
    demo_job    : FB_Executor;
    recipro_moving  : ARRAY [1..2, 1..10] OF FutureMCMoveAbsolute;
    _job_temp   : I_Job;				// Parallel jobコンテナのジョブへの参照変数
	i : UDINT;
	
	state : UDINT;
	fb_power : MC_Power;
	runner : FB_TaskRunner(ContainerType.PARALLEL_QUEUE);
	option : ST_MoveOptions;
END_VAR


IF NOT init THEN
    demo_job.create_container(ContainerType.BATCH, 'DEMO_JOB');
	
    FOR i := 1 TO 10 DO
		_job_temp := demo_job.children.create_container(ContainerType.PARALLEL,'Blending move container');
        IF i mod 2 > 0 THEN
            recipro_moving[1, i].set_parameters(GVL.axis1,500,600,0,0,0,MC_BufferMode.MC_Aborting);
			recipro_moving[1, i].future_name := 'Move +500 deg, 600 deg/s';
			recipro_moving[2, i].set_parameters(GVL.axis1,1000,50,0,0,0,MC_BufferMode.MC_BlendingNext);
			recipro_moving[2, i].future_name := 'Move +1000 deg, 50 deg/s';
        ELSE
            recipro_moving[1, i].set_parameters(GVL.axis1,500,600,0,0,0,MC_BufferMode.MC_Aborting);
			recipro_moving[1, i].future_name := 'Move +500 deg, 600 deg/s';
			recipro_moving[2, i].set_parameters(GVL.axis1,0,50,0,0,0,MC_BufferMode.MC_BlendingNext);
			recipro_moving[2, i].future_name := 'Move +0 deg, 50 deg/s';
        END_IF
        _job_temp.children.spawn_job(recipro_moving[1, i]);        
        _job_temp.children.spawn_job(recipro_moving[2, i]);        
		_job_temp := demo_job.children.append_job(_job_temp);
    END_FOR
    init := TRUE;
END_IF


CASE state OF
	0:
		fb_power(
			Axis:= GVL.axis1, 
			Enable:= TRUE, 
			Enable_Positive:= TRUE, 
			Enable_Negative:= TRUE, 
			Override:= 100 
		);
		IF fb_power.Status = TRUE THEN
			state := 1;
		END_IF
	1:
		runner.append_job(demo_job);
		state := 2;
	2:
		IF demo_job.ready THEN
			demo_job.start();
		END_IF
		IF demo_job.done THEN
			state := 3;
		END_IF
	3:
		fb_power(
			Axis:= GVL.axis1, 
			Enable:= FALSE, 
			Enable_Positive:= FALSE, 
			Enable_Negative:= FALSE, 
			Override:= 100 
		);
END_CASE

runner();

END_PROGRAM

// ---- POUs/model/activities/FutureCounterBlinkCreator.TcPOU
FUNCTION_BLOCK FutureCounterBlinkCreator IMPLEMENTS I_TaskCreator
VAR_INPUT
END_VAR
VAR_OUTPUT
END_VAR
VAR
	_target_count: UINT;
	_count_trigger: REFERENCE TO BOOL;
	_output: REFERENCE TO BOOL;
	_error_test :BOOL;
END_VAR

{warning 'add method implementation '}
METHOD create_future : I_Future
VAR_INPUT
	future_name :STRING;
END_VAR
VAR
	_p_future : POINTER TO FutureCounterBlink;
END_VAR
_p_future := __NEW(FutureCounterBlink);
_p_future^.future_name := future_name;
_p_future^.set_parameter(_target_count, _count_trigger, _output);
_p_future^.error_test := _error_test;
create_future := _p_future^;
END_METHOD

{warning 'add method implementation '}
METHOD destroy_future : I_Future
VAR_INPUT
	future : I_Future;
END_VAR
VAR
	_p_future : POINTER TO FutureCounterBlink;
END_VAR
IF __QUERYPOINTER(future, _p_future) THEN
	__DELETE(_p_future);
	IF _p_future = 0  THEN
		destroy_future := 0;
	END_IF
END_IF
END_METHOD

METHOD set_options : BOOL
VAR_INPUT
	error_test: BOOL;
END_VAR
_error_test := error_test;
END_METHOD

METHOD set_parameter : BOOL
VAR_INPUT
	target_count: UINT;
	count_trigger : REFERENCE TO BOOL;
	output		: REFERENCE TO BOOL;
END_VAR
_count_trigger REF= count_trigger;
_output REF= output;
_target_count := target_count;
END_METHOD

END_FUNCTION_BLOCK

// ---- POUs/model/activities/FutureCounterBlink.TcPOU
{attribute 'enable_dynamic_creation'}
FUNCTION_BLOCK FutureCounterBlink EXTENDS FB_AbstructFuture
VAR_INPUT
END_VAR
VAR_OUTPUT
END_VAR
VAR
	process_timer: TON;
	blink_timer: TON;
	_counter :UINT;
	_error_id :HRESULT;
	_target_count: UINT;
	_count_trigger: REFERENCE TO BOOL;
	_output: REFERENCE TO BOOL;
	_error_test :BOOL;
END_VAR

METHOD abort : BOOL
// The warning can be disabled here as the user is aware of the risk that the reference may not be valid by checking its validity
{warning disable C0371}
// Checking the VAR_IN_OUT reference, leave the current method in case of invalid reference
IF NOT __ISVALIDREF(_output) THEN
     RETURN;
END_IF

_output := FALSE;
abort := TRUE;

// The warning may be restored at the end of the access area
{warning restore C0371}
END_METHOD

PROPERTY counter : UINT
GET
counter := _counter;
END_GET
END_PROPERTY

METHOD error_reset : BOOL // Must be overrided if future has any errors.
_error_test := FALSE;
_error_id := 0;
error_reset := TRUE;
END_METHOD

PROPERTY error_test : BOOL
SET
_error_test := error_test;
END_SET
END_PROPERTY

METHOD execute : BOOL
VAR_INPUT
END_VAR
VAR_INST
	input_memory :BOOL;
END_VAR
// The warning can be disabled here as the user is aware of the risk that the reference may not be valid by checking its validity
{warning disable C0371}
// Checking the VAR_IN_OUT reference, leave the current method in case of invalid reference
IF NOT __ISVALIDREF(_output) OR NOT __ISVALIDREF(_count_trigger) THEN
	_error_id := 1;
     RETURN;
END_IF

IF _error_test THEN
	_error_id := 9;
	execute := TRUE;
END_IF

_output := TRUE;
IF _count_trigger AND NOT input_memory THEN
	_counter := _counter + 1;
END_IF
input_memory := _count_trigger;
IF _counter > _target_count THEN
	execute := TRUE;
END_IF

// The warning may be restored at the end of the access area
{warning restore C0371}
END_METHOD

METHOD init : BOOL
VAR_INPUT
END_VAR
// The warning can be disabled here as the user is aware of the risk that the reference may not be valid by checking its validity
{warning disable C0371}
// Checking the VAR_IN_OUT reference, leave the current method in case of invalid reference
IF NOT __ISVALIDREF(_output) THEN
	_error_id := 1;
     RETURN;
END_IF

_output := FALSE;
process_timer(IN := FALSE);
blink_timer(IN := FALSE);
_counter := 0;
init := TRUE;

// The warning may be restored at the end of the access area
{warning restore C0371}
END_METHOD

PROPERTY nErrorID : HRESULT
GET
nErrorID := _error_id;
END_GET
END_PROPERTY

METHOD quit : BOOL
THIS^.init();
quit := TRUE;
END_METHOD

METHOD set_options : BOOL
VAR_INPUT
	error_test: BOOL;
END_VAR
_error_test := error_test;
END_METHOD

METHOD set_parameter : BOOL
VAR_INPUT
	target_count: UINT;
	count_trigger : REFERENCE TO BOOL;
	output		: REFERENCE TO BOOL;
END_VAR
_count_trigger REF= count_trigger;
_output REF= output;
_target_count := target_count;
END_METHOD

END_FUNCTION_BLOCK

// ---- POUs/model/activities/FutureMCGearIn.TcPOU
{attribute 'enable_dynamic_creation'}
FUNCTION_BLOCK FutureMCGearIn EXTENDS FB_AbstructFuture
VAR_INPUT
END_VAR
VAR_OUTPUT
END_VAR
VAR
	_fb_gear_in	: MC_GearIn;
	_mc_reset	: MC_Reset;
	_axis_main: REFERENCE TO AXIS_REF;
	_axis_sub: REFERENCE TO AXIS_REF;
	_ratio_numerator	: MC_LREAL := 1;
	_ratio_denominator	: UINT := 1;
	_acceleration: MC_LREAL;
	_deceleration: MC_LREAL;
	_jerk		: MC_LREAL;
	_option : ST_GearInOptions;
	_buffer_mode : MC_BufferMode;
	_error_id :HRESULT;
	_exec_state : UDINT;
	_reset_state : UDINT;
END_VAR

